SPLINE
SPL {X  -160.133, Y  +702.956, Z    +0.000, E1   -19.806, E3 +400827.881}
SPL {X  -161.979, Y  +690.023, Z    +0.000, E1   -12.991, E3 +400830.798}
SPL {X  -162.641, Y  +681.139, Z    +0.000, E1    -7.893, E3 +400832.889}
SPL {X  -162.815, Y  +674.833, Z    +0.000, E1    -4.093, E3 +400830.505}
SPL {X  -162.820, Y  +669.862, Z    +0.000, E1    -0.751, E3 +400833.723}
SPL {X  -162.820, Y  +665.790, Z    +0.000, E1    +2.338, E3 +400833.096}
SPL {X  -162.820, Y  +660.758, Z    +0.000, E1    +6.523, E3 +400833.197}
SPL {X  -162.820, Y  +655.722, Z    +0.000, E1   +11.608, E3 +400829.570}
SPL {X  -162.820, Y  +648.706, Z    +0.000, E1   +17.761, E3 +400833.112}
SPL {X  -162.820, Y  +635.926, Z    +0.000, E1   +28.192, E3 +400837.939}
SPL {X  -162.820, Y  +621.673, Z    +0.000, E1   +34.265, E3 +400854.297}
SPL {X  -162.820, Y  +609.002, Z    +0.000, E1   +38.458, E3 +400867.518}
SPL {X  -162.820, Y  +596.392, Z    +0.000, E1   +37.895, E3 +400900.987}
ENDSPLINE

SPLINE
SPL {X  -162.820, Y  +601.432, Z    +0.000, E1   +34.026, E3 +400910.285}
ENDSPLINE

SPLINE
SPL {X  -162.820, Y  +597.570, Z    +0.000, E1   +33.919, E3 +400923.183}
SPL {X  -162.820, Y  +592.692, Z    +0.000, E1   +33.779, E3 +400939.074}
SPL {X  -162.820, Y  +588.795, Z    +0.000, E1   +33.876, E3 +400950.511}
SPL {X  -162.820, Y  +585.519, Z    +0.000, E1   +33.888, E3 +400960.596}
SPL {X  -162.820, Y  +582.066, Z    +0.000, E1   +33.857, E3 +400971.530}
SPL {X  -162.820, Y  +577.919, Z    +0.000, E1   +33.841, E3 +400984.583}
SPL {X  -162.820, Y  +573.566, Z    +0.000, E1   +33.899, E3 +400997.658}
SPL {X  -162.820, Y  +569.298, Z    +0.000, E1   +33.851, E3 +401011.300}
SPL {X  -162.820, Y  +565.024, Z    +0.000, E1   +33.872, E3 +401024.355}
SPL {X  -162.820, Y  +560.226, Z    +0.000, E1   +33.868, E3 +401039.449}
SPL {X  -162.820, Y  +556.206, Z    +0.000, E1   +33.843, E3 +401051.849}
SPL {X  -162.820, Y  +553.486, Z    +0.000, E1   +33.777, E3 +401060.795}
SPL {X  -162.820, Y  +549.726, Z    +0.000, E1   +33.905, E3 +401071.650}
SPL {X  -162.820, Y  +545.760, Z    +0.000, E1   +33.901, E3 +401084.046}
SPL {X  -162.820, Y  +541.668, Z    +0.000, E1   +33.787, E3 +401097.446}
SPL {X  -162.820, Y  +537.061, Z    +0.000, E1   +33.897, E3 +401111.104}
SPL {X  -162.820, Y  +532.164, Z    +0.000, E1   +33.861, E3 +401126.578}
SPL {X  -162.820, Y  +528.475, Z    +0.000, E1   +33.876, E3 +401137.746}
SPL {X  -162.820, Y  +524.900, Z    +0.000, E1   +33.820, E3 +401149.405}
SPL {X  -162.820, Y  +520.532, Z    +0.000, E1   +33.805, E3 +401162.973}
SPL {X  -162.820, Y  +515.754, Z    +0.000, E1   +33.911, E3 +401177.309}
SPL {X  -162.820, Y  +510.207, Z    +0.000, E1   +33.879, E3 +401194.689}
SPL {X  -162.820, Y  +504.570, Z    +0.000, E1   +33.876, E3 +401212.269}
SPL {X  -162.820, Y  +498.875, Z    +0.000, E1   +34.747, E3 +401223.970}
SPL {X  -162.820, Y  +481.122, Z    +0.000, E1   +41.279, E3 +401231.121}
SPL {X  -162.820, Y  +477.698, Z    +0.000, E1   +40.353, E3 +401245.177}
SPL {X  -162.820, Y  +473.851, Z    +0.000, E1   +39.059, E3 +401262.569}
SPL {X  -162.820, Y  +470.157, Z    +0.000, E1   +38.016, E3 +401278.506}
SPL {X  -162.820, Y  +467.216, Z    +0.000, E1   +37.215, E3 +401291.267}
SPL {X  -162.820, Y  +462.598, Z    +0.000, E1   +37.325, E3 +401303.221}
SPL {X  -162.820, Y  +459.177, Z    +0.000, E1   +37.207, E3 +401313.249}
SPL {X  -162.820, Y  +453.939, Z    +0.000, E1   +37.397, E3 +401326.601}
SPL {X  -162.820, Y  +448.311, Z    +0.000, E1   +37.333, E3 +401342.262}
SPL {X  -162.820, Y  +443.351, Z    +0.000, E1   +37.335, E3 +401355.792}
SPL {X  -162.820, Y  +438.727, Z    +0.000, E1   +37.289, E3 +401368.664}
SPL {X  -162.820, Y  +434.320, Z    +0.000, E1   +37.343, E3 +401380.374}
SPL {X  -162.820, Y  +430.091, Z    +0.000, E1   +37.424, E3 +401391.374}
SPL {X  -162.820, Y  +426.177, Z    +0.000, E1   +37.250, E3 +401403.197}
SPL {X  -162.820, Y  +420.241, Z    +0.000, E1   +37.355, E3 +401418.903}
SPL {X  -162.820, Y  +415.595, Z    +0.000, E1   +37.375, E3 +401431.243}
SPL {X  -162.820, Y  +411.860, Z    +0.000, E1   +37.402, E3 +401441.346}
SPL {X  -162.820, Y  +407.726, Z    +0.000, E1   +37.291, E3 +401453.294}
SPL {X  -162.820, Y  +403.543, Z    +0.000, E1   +37.305, E3 +401464.639}
SPL {X  -162.820, Y  +399.300, Z    +0.000, E1   +37.355, E3 +401475.924}
SPL {X  -162.820, Y  +395.182, Z    +0.000, E1   +37.347, E3 +401487.213}
SPL {X  -162.820, Y  +390.797, Z    +0.000, E1   +37.358, E3 +401499.125}
SPL {X  -162.820, Y  +386.671, Z    +0.000, E1   +37.363, E3 +401510.306}
SPL {X  -162.820, Y  +382.174, Z    +0.000, E1   +37.329, E3 +401522.883}
SPL {X  -162.785, Y  +377.133, Z    +0.000, E1   +37.299, E3 +401536.813}
SPL {X  -162.576, Y  +371.586, Z    +0.000, E1   +37.322, E3 +401551.925}
SPL {X  -162.256, Y  +366.963, Z    +0.000, E1   +37.251, E3 +401564.814}
SPL {X  -161.920, Y  +363.407, Z    +0.000, E1   +37.164, E3 +401575.099}
SPL {X  -161.341, Y  +358.603, Z    +0.000, E1   +37.117, E3 +401588.579}
SPL {X  -160.616, Y  +353.801, Z    +0.000, E1   +36.942, E3 +401602.744}
SPL {X  -159.837, Y  +349.474, Z    +0.000, E1   +36.824, E3 +401615.188}
SPL {X  -159.171, Y  +346.224, Z    +0.000, E1   +36.747, E3 +401624.464}
SPL {X  -158.248, Y  +342.188, Z    +0.000, E1   +36.583, E3 +401636.627}
SPL {X  -153.520, Y  +326.260, Z    +0.000, E1   +41.363, E3 +401649.279}
SPL {X  -150.942, Y  +319.452, Z    +0.000, E1   +36.529, E3 +401705.636}
ENDSPLINE

SPLINE
SPL {X  -159.264, Y  +346.659, Z    +0.000, E1   +22.083, E3 +401746.211}
SPL {X  -161.245, Y  +357.907, Z    +0.000, E1   +16.095, E3 +401759.643}
SPL {X  -162.697, Y  +374.161, Z    +0.000, E1    +7.119, E3 +401757.633}
SPL {X  -162.820, Y  +380.878, Z    +0.000, E1    +2.854, E3 +401760.464}
SPL {X  -162.820, Y  +385.313, Z    +0.000, E1    -0.228, E3 +401760.244}
SPL {X  -162.820, Y  +389.965, Z    +0.000, E1    -3.918, E3 +401759.613}
SPL {X  -162.820, Y  +394.532, Z    +0.000, E1    -7.849, E3 +401761.161}
SPL {X  -162.820, Y  +400.765, Z    +0.000, E1   -14.108, E3 +401758.628}
SPL {X  -162.820, Y  +411.829, Z    +0.000, E1   -24.195, E3 +401760.705}
SPL {X  -162.820, Y  +434.900, Z    +0.000, E1   -34.666, E3 +401788.070}
SPL {X  -162.820, Y  +465.440, Z    +0.000, E1   -41.264, E3 +401829.377}
ENDSPLINE

SPLINE
SPL {X  -162.820, Y  +460.175, Z    +0.000, E1   -36.098, E3 +401847.177}
ENDSPLINE

SPLINE
SPL {X  -162.820, Y  +465.690, Z    +0.000, E1   -36.140, E3 +401862.491}
SPL {X  -162.820, Y  +470.432, Z    +0.000, E1   -36.100, E3 +401876.374}
SPL {X  -162.820, Y  +475.701, Z    +0.000, E1   -36.157, E3 +401891.001}
SPL {X  -162.820, Y  +479.954, Z    +0.000, E1   -36.086, E3 +401903.542}
SPL {X  -162.820, Y  +485.438, Z    +0.000, E1   -36.112, E3 +401919.260}
SPL {X  -162.820, Y  +490.843, Z    +0.000, E1   -36.087, E3 +401934.673}
SPL {X  -162.820, Y  +494.712, Z    +0.000, E1   -36.164, E3 +401945.185}
SPL {X  -162.820, Y  +497.796, Z    +0.000, E1   -36.022, E3 +401954.891}
SPL {X  -162.820, Y  +502.146, Z    +0.000, E1   -36.123, E3 +401966.760}
SPL {X  -162.820, Y  +505.688, Z    +0.000, E1   -36.050, E3 +401977.242}
SPL {X  -162.820, Y  +509.364, Z    +0.000, E1   -36.084, E3 +401987.613}
SPL {X  -162.820, Y  +513.393, Z    +0.000, E1   -36.179, E3 +401998.469}
SPL {X  -162.820, Y  +516.436, Z    +0.000, E1   -36.094, E3 +402007.665}
SPL {X  -162.820, Y  +520.482, Z    +0.000, E1   -36.096, E3 +402019.296}
SPL {X  -162.820, Y  +524.107, Z    +0.000, E1   -36.045, E3 +402029.880}
SPL {X  -162.820, Y  +527.962, Z    +0.000, E1   -36.074, E3 +402040.813}
SPL {X  -162.820, Y  +532.253, Z    +0.000, E1   -36.170, E3 +402052.402}
SPL {X  -162.820, Y  +536.031, Z    +0.000, E1   -36.058, E3 +402063.940}
SPL {X  -162.820, Y  +541.179, Z    +0.000, E1   -36.085, E3 +402078.581}
SPL {X  -162.820, Y  +546.355, Z    +0.000, E1   -36.114, E3 +402093.125}
SPL {X  -162.820, Y  +551.776, Z    +0.000, E1   -36.108, E3 +402108.759}
SPL {X  -162.820, Y  +558.272, Z    +0.000, E1   -36.170, E3 +402126.967}
SPL {X  -162.820, Y  +562.721, Z    +0.000, E1   -36.046, E3 +402140.192}
SPL {X  -162.820, Y  +566.500, Z    +0.000, E1   -36.073, E3 +402150.924}
SPL {X  -162.820, Y  +570.319, Z    +0.000, E1   -36.045, E3 +402161.953}
SPL {X  -162.820, Y  +573.265, Z    +0.000, E1   -36.071, E3 +402170.189}
SPL {X  -162.820, Y  +576.887, Z    +0.000, E1   -36.084, E3 +402180.547}
SPL {X  -162.820, Y  +581.763, Z    +0.000, E1   -36.093, E3 +402194.484}
SPL {X  -162.820, Y  +586.693, Z    +0.000, E1   -36.086, E3 +402208.589}
SPL {X  -162.820, Y  +591.665, Z    +0.000, E1   -36.045, E3 +402223.117}
SPL {X  -162.820, Y  +597.399, Z    +0.000, E1   -36.147, E3 +402238.880}
SPL {X  -162.820, Y  +602.243, Z    +0.000, E1   -36.085, E3 +402253.026}
SPL {X  -162.820, Y  +605.848, Z    +0.000, E1   -36.070, E3 +402263.348}
SPL {X  -162.820, Y  +609.375, Z    +0.000, E1   -36.084, E3 +402273.398}
SPL {X  -162.820, Y  +612.959, Z    +0.000, E1   -36.034, E3 +402283.918}
SPL {X  -162.820, Y  +616.897, Z    +0.000, E1   -36.061, E3 +402295.066}
SPL {X  -162.820, Y  +621.516, Z    +0.000, E1   -36.072, E3 +402308.265}
SPL {X  -162.820, Y  +626.243, Z    +0.000, E1   -36.105, E3 +402321.508}
SPL {X  -162.820, Y  +630.571, Z    +0.000, E1   -36.057, E3 +402334.210}
SPL {X  -162.820, Y  +634.189, Z    +0.000, E1   -36.065, E3 +402344.403}
SPL {X  -162.820, Y  +638.473, Z    +0.000, E1   -36.098, E3 +402356.640}
SPL {X  -162.820, Y  +642.832, Z    +0.000, E1   -36.091, E3 +402368.966}
SPL {X  -162.820, Y  +646.320, Z    +0.000, E1   -36.078, E3 +402379.073}
SPL {X  -162.820, Y  +649.997, Z    +0.000, E1   -36.000, E3 +402390.044}
SPL {X  -162.820, Y  +655.571, Z    +0.000, E1   -36.141, E3 +402405.378}
SPL {X  -162.820, Y  +661.560, Z    +0.000, E1   -36.068, E3 +402422.806}
SPL {X  -162.820, Y  +667.641, Z    +0.000, E1   -36.092, E3 +402440.187}
SPL {X  -162.820, Y  +673.415, Z    +0.000, E1   -36.053, E3 +402456.777}
SPL {X  -162.761, Y  +677.889, Z    +0.000, E1   -36.122, E3 +402469.095}
SPL {X  -162.577, Y  +682.401, Z    +0.000, E1   -36.021, E3 +402482.712}
SPL {X  -162.187, Y  +687.846, Z    +0.000, E1   -36.007, E3 +402498.381}
SPL {X  -161.667, Y  +692.839, Z    +0.000, E1   -35.918, E3 +402513.146}
SPL {X  -161.078, Y  +697.256, Z    +0.000, E1   -35.797, E3 +402526.482}
SPL {X  -160.313, Y  +701.964, Z    +0.000, E1   -35.709, E3 +402540.558}
SPL {X  -159.317, Y  +707.091, Z    +0.000, E1   -35.482, E3 +402556.582}
SPL {X  -158.510, Y  +710.714, Z    +0.000, E1   -35.230, E3 +402568.293}
SPL {X  -155.037, Y  +723.239, Z    +0.000, E1   -39.382, E3 +402577.389}
SPL {X  -152.141, Y  +731.494, Z    +0.000, E1   -35.181, E3 +402636.195}
ENDSPLINE

SPLINE
SPL {X  -160.133, Y  +702.956, Z    +0.000, E1   -19.806, E3 +402679.733}
SPL {X  -161.979, Y  +690.023, Z    +0.000, E1   -12.991, E3 +402682.649}
SPL {X  -162.641, Y  +681.139, Z    +0.000, E1    -7.893, E3 +402684.741}
SPL {X  -162.815, Y  +674.833, Z    +0.000, E1    -4.093, E3 +402682.357}
SPL {X  -162.820, Y  +669.862, Z    +0.000, E1    -0.751, E3 +402685.575}
SPL {X  -162.820, Y  +664.572, Z    +0.000, E1    +3.252, E3 +402685.389}
SPL {X  -162.820, Y  +657.781, Z    +0.000, E1    +9.391, E3 +402683.212}
SPL {X  -162.820, Y  +648.706, Z    +0.000, E1   +17.761, E3 +402684.964}
SPL {X  -162.820, Y  +635.926, Z    +0.000, E1   +28.192, E3 +402689.791}
SPL {X  -162.820, Y  +621.673, Z    +0.000, E1   +34.265, E3 +402706.149}
SPL {X  -162.820, Y  +601.185, Z    +0.000, E1   +39.430, E3 +402732.727}
SPL {X  -162.820, Y  +599.927, Z    +0.000, E1   +35.241, E3 +402759.305}
SPL {X  -162.820, Y  +597.570, Z    +0.000, E1   +33.919, E3 +402775.034}
SPL {X  -162.820, Y  +592.692, Z    +0.000, E1   +33.779, E3 +402790.926}
SPL {X  -162.820, Y  +588.795, Z    +0.000, E1   +33.876, E3 +402802.363}
SPL {X  -162.820, Y  +584.646, Z    +0.000, E1   +33.882, E3 +402815.327}
SPL {X  -162.820, Y  +579.919, Z    +0.000, E1   +33.857, E3 +402830.115}
SPL {X  -162.820, Y  +574.615, Z    +0.000, E1   +33.920, E3 +402846.289}
SPL {X  -162.820, Y  +570.335, Z    +0.000, E1   +33.821, E3 +402859.995}
SPL {X  -162.820, Y  +565.901, Z    +0.000, E1   +33.889, E3 +402873.515}
SPL {X  -162.820, Y  +562.173, Z    +0.000, E1   +33.897, E3 +402884.806}
SPL {X  -162.820, Y  +558.179, Z    +0.000, E1   +33.857, E3 +402897.742}
SPL {X  -162.820, Y  +553.486, Z    +0.000, E1   +33.777, E3 +402912.647}
SPL {X  -162.820, Y  +548.576, Z    +0.000, E1   +33.950, E3 +402926.929}
SPL {X  -162.820, Y  +544.808, Z    +0.000, E1   +33.827, E3 +402939.191}
SPL {X  -162.820, Y  +541.668, Z    +0.000, E1   +33.787, E3 +402949.297}
SPL {X  -162.820, Y  +538.174, Z    +0.000, E1   +33.865, E3 +402959.587}
SPL {X  -162.820, Y  +534.943, Z    +0.000, E1   +33.919, E3 +402969.327}
SPL {X  -162.820, Y  +531.459, Z    +0.000, E1   +33.783, E3 +402980.984}
SPL {X  -162.820, Y  +528.475, Z    +0.000, E1   +33.876, E3 +402989.598}
SPL {X  -162.820, Y  +524.900, Z    +0.000, E1   +33.820, E3 +403001.257}
SPL {X  -162.820, Y  +520.532, Z    +0.000, E1   +33.805, E3 +403014.825}
SPL {X  -162.820, Y  +516.814, Z    +0.000, E1   +33.917, E3 +403025.661}
SPL {X  -162.820, Y  +512.685, Z    +0.000, E1   +33.830, E3 +403039.103}
SPL {X  -162.820, Y  +508.888, Z    +0.000, E1   +33.871, E3 +403050.518}
SPL {X  -162.820, Y  +505.651, Z    +0.000, E1   +33.839, E3 +403060.835}
SPL {X  -162.820, Y  +500.931, Z    +0.000, E1   +34.256, E3 +403072.709}
SPL {X  -162.820, Y  +481.122, Z    +0.000, E1   +41.279, E3 +403082.973}
SPL {X  -162.820, Y  +477.698, Z    +0.000, E1   +40.353, E3 +403097.029}
SPL {X  -162.820, Y  +474.538, Z    +0.000, E1   +39.267, E3 +403111.205}
SPL {X  -162.820, Y  +472.097, Z    +0.000, E1   +38.411, E3 +403122.748}
SPL {X  -162.820, Y  +469.308, Z    +0.000, E1   +37.839, E3 +403133.553}
SPL {X  -162.820, Y  +467.216, Z    +0.000, E1   +37.215, E3 +403143.119}
SPL {X  -162.820, Y  +462.598, Z    +0.000, E1   +37.325, E3 +403155.073}
SPL {X  -162.820, Y  +457.832, Z    +0.000, E1   +37.294, E3 +403168.360}
SPL {X  -162.820, Y  +452.986, Z    +0.000, E1   +37.368, E3 +403181.094}
SPL {X  -162.820, Y  +448.311, Z    +0.000, E1   +37.333, E3 +403194.114}
SPL {X  -162.820, Y  +443.351, Z    +0.000, E1   +37.335, E3 +403207.643}
SPL {X  -162.820, Y  +438.727, Z    +0.000, E1   +37.289, E3 +403220.516}
SPL {X  -162.820, Y  +434.320, Z    +0.000, E1   +37.343, E3 +403232.226}
SPL {X  -162.820, Y  +430.091, Z    +0.000, E1   +37.424, E3 +403243.226}
SPL {X  -162.820, Y  +426.177, Z    +0.000, E1   +37.250, E3 +403255.048}
SPL {X  -162.820, Y  +421.391, Z    +0.000, E1   +37.346, E3 +403267.512}
SPL {X  -162.820, Y  +416.811, Z    +0.000, E1   +37.348, E3 +403280.046}
SPL {X  -162.820, Y  +411.860, Z    +0.000, E1   +37.402, E3 +403293.198}
SPL {X  -162.820, Y  +407.726, Z    +0.000, E1   +37.291, E3 +403305.146}
SPL {X  -162.820, Y  +403.543, Z    +0.000, E1   +37.305, E3 +403316.491}
SPL {X  -162.820, Y  +399.300, Z    +0.000, E1   +37.355, E3 +403327.776}
SPL {X  -162.820, Y  +395.182, Z    +0.000, E1   +37.347, E3 +403339.065}
SPL {X  -162.820, Y  +390.797, Z    +0.000, E1   +37.358, E3 +403350.977}
SPL {X  -162.820, Y  +385.307, Z    +0.000, E1   +37.364, E3 +403366.057}
SPL {X  -162.820, Y  +380.796, Z    +0.000, E1   +37.334, E3 +403378.343}
SPL {X  -162.785, Y  +377.133, Z    +0.000, E1   +37.299, E3 +403388.664}
SPL {X  -162.623, Y  +372.484, Z    +0.000, E1   +37.337, E3 +403401.104}
SPL {X  -162.331, Y  +367.894, Z    +0.000, E1   +37.251, E3 +403414.217}
SPL {X  -161.920, Y  +363.407, Z    +0.000, E1   +37.164, E3 +403426.951}
SPL {X  -161.341, Y  +358.603, Z    +0.000, E1   +37.117, E3 +403440.431}
SPL {X  -160.616, Y  +353.801, Z    +0.000, E1   +36.942, E3 +403454.595}
SPL {X  -159.837, Y  +349.474, Z    +0.000, E1   +36.824, E3 +403467.040}
SPL {X  -158.862, Y  +344.820, Z    +0.000, E1   +36.732, E3 +403480.402}
SPL {X  -157.959, Y  +341.011, Z    +0.000, E1   +36.448, E3 +403492.299}
SPL {X  -154.495, Y  +329.104, Z    +0.000, E1   +40.891, E3 +403497.182}
SPL {X  -152.543, Y  +323.569, Z    +0.000, E1   +41.772, E3 +403504.938}
SPL {X  -150.942, Y  +319.452, Z    +0.000, E1   +36.529, E3 +403557.488}
ENDSPLINE

SPLINE
SPL {X  -159.264, Y  +346.659, Z    +0.000, E1   +22.083, E3 +403598.062}
SPL {X  -161.245, Y  +357.907, Z    +0.000, E1   +16.095, E3 +403611.495}
SPL {X  -162.697, Y  +374.161, Z    +0.000, E1    +7.119, E3 +403609.485}
SPL {X  -162.820, Y  +380.878, Z    +0.000, E1    +2.854, E3 +403612.316}
SPL {X  -162.820, Y  +385.313, Z    +0.000, E1    -0.228, E3 +403612.096}
SPL {X  -162.820, Y  +389.965, Z    +0.000, E1    -3.918, E3 +403611.465}
SPL {X  -162.820, Y  +394.532, Z    +0.000, E1    -7.849, E3 +403613.013}
SPL {X  -162.820, Y  +400.765, Z    +0.000, E1   -14.108, E3 +403610.480}
SPL {X  -162.820, Y  +411.829, Z    +0.000, E1   -24.195, E3 +403612.557}
SPL {X  -162.820, Y  +434.900, Z    +0.000, E1   -34.666, E3 +403639.922}
SPL {X  -162.820, Y  +465.440, Z    +0.000, E1   -41.264, E3 +403681.229}
ENDSPLINE

SPLINE
SPL {X  -162.820, Y  +460.175, Z    +0.000, E1   -36.098, E3 +403699.029}
ENDSPLINE

SPLINE
SPL {X  -162.820, Y  +465.690, Z    +0.000, E1   -36.140, E3 +403714.343}
SPL {X  -162.820, Y  +470.432, Z    +0.000, E1   -36.100, E3 +403728.226}
SPL {X  -162.820, Y  +475.701, Z    +0.000, E1   -36.157, E3 +403742.853}
SPL {X  -162.820, Y  +479.954, Z    +0.000, E1   -36.086, E3 +403755.393}
SPL {X  -162.820, Y  +485.438, Z    +0.000, E1   -36.112, E3 +403771.112}
SPL {X  -162.820, Y  +490.843, Z    +0.000, E1   -36.087, E3 +403786.525}
SPL {X  -162.820, Y  +494.712, Z    +0.000, E1   -36.164, E3 +403797.037}
SPL {X  -162.820, Y  +497.796, Z    +0.000, E1   -36.022, E3 +403806.743}
SPL {X  -162.820, Y  +502.146, Z    +0.000, E1   -36.123, E3 +403818.612}
SPL {X  -162.820, Y  +505.688, Z    +0.000, E1   -36.050, E3 +403829.094}
SPL {X  -162.820, Y  +509.364, Z    +0.000, E1   -36.084, E3 +403839.465}
SPL {X  -162.820, Y  +513.393, Z    +0.000, E1   -36.179, E3 +403850.321}
SPL {X  -162.820, Y  +516.436, Z    +0.000, E1   -36.094, E3 +403859.517}
SPL {X  -162.820, Y  +520.482, Z    +0.000, E1   -36.096, E3 +403871.148}
SPL {X  -162.820, Y  +524.107, Z    +0.000, E1   -36.045, E3 +403881.732}
SPL {X  -162.820, Y  +527.962, Z    +0.000, E1   -36.074, E3 +403892.665}
SPL {X  -162.820, Y  +532.253, Z    +0.000, E1   -36.170, E3 +403904.254}
SPL {X  -162.820, Y  +536.031, Z    +0.000, E1   -36.058, E3 +403915.792}
SPL {X  -162.820, Y  +541.179, Z    +0.000, E1   -36.085, E3 +403930.433}
SPL {X  -162.820, Y  +546.355, Z    +0.000, E1   -36.114, E3 +403944.977}
SPL {X  -162.820, Y  +551.776, Z    +0.000, E1   -36.108, E3 +403960.611}
SPL {X  -162.820, Y  +558.272, Z    +0.000, E1   -36.170, E3 +403978.819}
SPL {X  -162.820, Y  +562.721, Z    +0.000, E1   -36.046, E3 +403992.044}
SPL {X  -162.820, Y  +566.500, Z    +0.000, E1   -36.073, E3 +404002.776}
SPL {X  -162.820, Y  +570.319, Z    +0.000, E1   -36.045, E3 +404013.804}
SPL {X  -162.820, Y  +573.265, Z    +0.000, E1   -36.071, E3 +404022.041}
SPL {X  -162.820, Y  +576.887, Z    +0.000, E1   -36.084, E3 +404032.399}
SPL {X  -162.820, Y  +581.763, Z    +0.000, E1   -36.093, E3 +404046.336}
SPL {X  -162.820, Y  +586.693, Z    +0.000, E1   -36.086, E3 +404060.441}
SPL {X  -162.820, Y  +591.665, Z    +0.000, E1   -36.045, E3 +404074.969}
SPL {X  -162.820, Y  +597.399, Z    +0.000, E1   -36.147, E3 +404090.732}
SPL {X  -162.820, Y  +602.243, Z    +0.000, E1   -36.085, E3 +404104.878}
SPL {X  -162.820, Y  +605.848, Z    +0.000, E1   -36.070, E3 +404115.199}
SPL {X  -162.820, Y  +609.375, Z    +0.000, E1   -36.084, E3 +404125.250}
SPL {X  -162.820, Y  +612.959, Z    +0.000, E1   -36.034, E3 +404135.770}
SPL {X  -162.820, Y  +616.897, Z    +0.000, E1   -36.061, E3 +404146.918}
SPL {X  -162.820, Y  +621.516, Z    +0.000, E1   -36.072, E3 +404160.117}
SPL {X  -162.820, Y  +626.243, Z    +0.000, E1   -36.105, E3 +404173.360}
SPL {X  -162.820, Y  +630.571, Z    +0.000, E1   -36.057, E3 +404186.062}
SPL {X  -162.820, Y  +634.189, Z    +0.000, E1   -36.065, E3 +404196.255}
SPL {X  -162.820, Y  +638.473, Z    +0.000, E1   -36.098, E3 +404208.492}
SPL {X  -162.820, Y  +642.832, Z    +0.000, E1   -36.091, E3 +404220.818}
SPL {X  -162.820, Y  +646.320, Z    +0.000, E1   -36.078, E3 +404230.925}
SPL {X  -162.820, Y  +649.997, Z    +0.000, E1   -36.000, E3 +404241.896}
SPL {X  -162.820, Y  +655.571, Z    +0.000, E1   -36.141, E3 +404257.230}
SPL {X  -162.820, Y  +661.560, Z    +0.000, E1   -36.068, E3 +404274.658}
SPL {X  -162.820, Y  +667.641, Z    +0.000, E1   -36.092, E3 +404292.039}
SPL {X  -162.820, Y  +673.415, Z    +0.000, E1   -36.053, E3 +404308.629}
SPL {X  -162.761, Y  +677.889, Z    +0.000, E1   -36.122, E3 +404320.947}
SPL {X  -162.577, Y  +682.401, Z    +0.000, E1   -36.021, E3 +404334.564}
SPL {X  -162.187, Y  +687.846, Z    +0.000, E1   -36.007, E3 +404350.233}
SPL {X  -161.667, Y  +692.839, Z    +0.000, E1   -35.918, E3 +404364.998}
SPL {X  -161.078, Y  +697.256, Z    +0.000, E1   -35.797, E3 +404378.334}
SPL {X  -160.313, Y  +701.964, Z    +0.000, E1   -35.709, E3 +404392.410}
SPL {X  -159.317, Y  +707.091, Z    +0.000, E1   -35.482, E3 +404408.433}
SPL {X  -158.510, Y  +710.714, Z    +0.000, E1   -35.230, E3 +404420.144}
SPL {X  -155.037, Y  +723.239, Z    +0.000, E1   -39.382, E3 +404429.241}
SPL {X  -152.141, Y  +731.494, Z    +0.000, E1   -35.181, E3 +404488.047}
ENDSPLINE

SPLINE
SPL {X  -152.670, Y  +730.088, Z    +0.000, E1   -30.916, E3 +404561.409}
SPL {X  -160.727, Y  +699.521, Z    +0.000, E1   -18.202, E3 +404527.692}
SPL {X  -161.979, Y  +690.023, Z    +0.000, E1   -12.991, E3 +404534.501}
SPL {X  -162.641, Y  +681.139, Z    +0.000, E1    -7.893, E3 +404536.593}
SPL {X  -162.820, Y  +673.062, Z    +0.000, E1    -2.992, E3 +404535.560}
SPL {X  -162.820, Y  +666.731, Z    +0.000, E1    +1.545, E3 +404537.190}
SPL {X  -162.820, Y  +660.758, Z    +0.000, E1    +6.523, E3 +404536.901}
SPL {X  -162.820, Y  +650.583, Z    +0.000, E1   +16.035, E3 +404535.873}
SPL {X  -162.820, Y  +629.267, Z    +0.000, E1   +31.872, E3 +404547.022}
SPL {X  -162.820, Y  +617.390, Z    +0.000, E1   +35.413, E3 +404563.951}
SPL {X  -162.820, Y  +596.392, Z    +0.000, E1   +37.895, E3 +404604.691}
ENDSPLINE

SPLINE
SPL {X  -162.820, Y  +601.432, Z    +0.000, E1   +34.026, E3 +404613.989}
ENDSPLINE

SPLINE
SPL {X  -162.820, Y  +597.570, Z    +0.000, E1   +33.919, E3 +404626.886}
SPL {X  -162.820, Y  +592.692, Z    +0.000, E1   +33.779, E3 +404642.778}
SPL {X  -162.820, Y  +588.795, Z    +0.000, E1   +33.876, E3 +404654.215}
SPL {X  -162.820, Y  +585.519, Z    +0.000, E1   +33.888, E3 +404664.300}
SPL {X  -162.820, Y  +582.066, Z    +0.000, E1   +33.857, E3 +404675.234}
SPL {X  -162.820, Y  +577.919, Z    +0.000, E1   +33.841, E3 +404688.287}
SPL {X  -162.820, Y  +573.566, Z    +0.000, E1   +33.899, E3 +404701.362}
SPL {X  -162.820, Y  +569.298, Z    +0.000, E1   +33.851, E3 +404715.003}
SPL {X  -162.820, Y  +563.983, Z    +0.000, E1   +33.916, E3 +404731.144}
SPL {X  -162.820, Y  +559.395, Z    +0.000, E1   +33.796, E3 +404746.025}
SPL {X  -162.820, Y  +554.453, Z    +0.000, E1   +33.841, E3 +404761.250}
SPL {X  -162.820, Y  +549.726, Z    +0.000, E1   +33.905, E3 +404775.353}
SPL {X  -162.820, Y  +545.760, Z    +0.000, E1   +33.901, E3 +404787.749}
SPL {X  -162.820, Y  +541.668, Z    +0.000, E1   +33.787, E3 +404801.149}
SPL {X  -162.820, Y  +538.174, Z    +0.000, E1   +33.865, E3 +404811.439}
SPL {X  -162.820, Y  +534.943, Z    +0.000, E1   +33.919, E3 +404821.179}
SPL {X  -162.820, Y  +530.273, Z    +0.000, E1   +33.855, E3 +404836.208}
SPL {X  -162.820, Y  +524.900, Z    +0.000, E1   +33.820, E3 +404853.109}
SPL {X  -162.820, Y  +520.532, Z    +0.000, E1   +33.805, E3 +404866.677}
SPL {X  -162.820, Y  +516.814, Z    +0.000, E1   +33.917, E3 +404877.513}
SPL {X  -162.820, Y  +512.685, Z    +0.000, E1   +33.830, E3 +404890.955}
SPL {X  -162.820, Y  +508.888, Z    +0.000, E1   +33.871, E3 +404902.370}
SPL {X  -162.820, Y  +505.651, Z    +0.000, E1   +33.839, E3 +404912.687}
SPL {X  -162.820, Y  +500.931, Z    +0.000, E1   +34.256, E3 +404924.561}
SPL {X  -162.820, Y  +481.122, Z    +0.000, E1   +41.279, E3 +404934.825}
SPL {X  -162.820, Y  +477.698, Z    +0.000, E1   +40.353, E3 +404948.881}
SPL {X  -162.820, Y  +474.538, Z    +0.000, E1   +39.267, E3 +404963.056}
SPL {X  -162.820, Y  +472.097, Z    +0.000, E1   +38.411, E3 +404974.600}
SPL {X  -162.820, Y  +469.308, Z    +0.000, E1   +37.839, E3 +404985.404}
SPL {X  -162.820, Y  +467.216, Z    +0.000, E1   +37.215, E3 +404994.971}
SPL {X  -162.820, Y  +462.598, Z    +0.000, E1   +37.325, E3 +405006.925}
SPL {X  -162.820, Y  +457.832, Z    +0.000, E1   +37.294, E3 +405020.212}
SPL {X  -162.820, Y  +452.986, Z    +0.000, E1   +37.368, E3 +405032.946}
SPL {X  -162.820, Y  +448.311, Z    +0.000, E1   +37.333, E3 +405045.966}
SPL {X  -162.820, Y  +443.351, Z    +0.000, E1   +37.335, E3 +405059.495}
SPL {X  -162.820, Y  +438.727, Z    +0.000, E1   +37.289, E3 +405072.368}
SPL {X  -162.820, Y  +434.320, Z    +0.000, E1   +37.343, E3 +405084.078}
SPL {X  -162.820, Y  +430.091, Z    +0.000, E1   +37.424, E3 +405095.078}
SPL {X  -162.820, Y  +426.177, Z    +0.000, E1   +37.250, E3 +405106.900}
SPL {X  -162.820, Y  +421.391, Z    +0.000, E1   +37.346, E3 +405119.364}
SPL {X  -162.820, Y  +416.811, Z    +0.000, E1   +37.348, E3 +405131.898}
SPL {X  -162.820, Y  +411.860, Z    +0.000, E1   +37.402, E3 +405145.050}
SPL {X  -162.820, Y  +407.726, Z    +0.000, E1   +37.291, E3 +405156.998}
SPL {X  -162.820, Y  +403.543, Z    +0.000, E1   +37.305, E3 +405168.343}
SPL {X  -162.820, Y  +399.300, Z    +0.000, E1   +37.355, E3 +405179.627}
SPL {X  -162.820, Y  +395.182, Z    +0.000, E1   +37.347, E3 +405190.917}
SPL {X  -162.820, Y  +390.797, Z    +0.000, E1   +37.358, E3 +405202.829}
SPL {X  -162.820, Y  +385.307, Z    +0.000, E1   +37.364, E3 +405217.908}
SPL {X  -162.820, Y  +380.796, Z    +0.000, E1   +37.334, E3 +405230.195}
SPL {X  -162.785, Y  +377.133, Z    +0.000, E1   +37.299, E3 +405240.516}
SPL {X  -162.623, Y  +372.484, Z    +0.000, E1   +37.337, E3 +405252.956}
SPL {X  -162.331, Y  +367.894, Z    +0.000, E1   +37.251, E3 +405266.069}
SPL {X  -161.920, Y  +363.407, Z    +0.000, E1   +37.164, E3 +405278.803}
SPL {X  -161.341, Y  +358.603, Z    +0.000, E1   +37.117, E3 +405292.283}
SPL {X  -160.616, Y  +353.801, Z    +0.000, E1   +36.942, E3 +405306.447}
SPL {X  -159.837, Y  +349.474, Z    +0.000, E1   +36.824, E3 +405318.891}
SPL {X  -158.862, Y  +344.820, Z    +0.000, E1   +36.732, E3 +405332.254}
SPL {X  -157.959, Y  +341.011, Z    +0.000, E1   +36.448, E3 +405344.151}
SPL {X  -154.495, Y  +329.104, Z    +0.000, E1   +40.891, E3 +405349.033}
SPL {X  -152.543, Y  +323.569, Z    +0.000, E1   +41.772, E3 +405356.790}
SPL {X  -150.942, Y  +319.452, Z    +0.000, E1   +36.529, E3 +405409.340}
ENDSPLINE

SPLINE
SPL {X  -159.264, Y  +346.659, Z    +0.000, E1   +22.083, E3 +405449.914}
SPL {X  -161.245, Y  +357.907, Z    +0.000, E1   +16.095, E3 +405463.347}
SPL {X  -162.746, Y  +375.590, Z    +0.000, E1    +6.280, E3 +405462.935}
SPL {X  -162.820, Y  +384.478, Z    +0.000, E1    +0.434, E3 +405463.605}
SPL {X  -162.820, Y  +389.965, Z    +0.000, E1    -3.918, E3 +405463.316}
SPL {X  -162.820, Y  +394.532, Z    +0.000, E1    -7.849, E3 +405464.865}
SPL {X  -162.820, Y  +400.765, Z    +0.000, E1   -14.108, E3 +405462.331}
SPL {X  -162.820, Y  +411.829, Z    +0.000, E1   -24.195, E3 +405464.409}
SPL {X  -162.820, Y  +434.900, Z    +0.000, E1   -34.666, E3 +405491.774}
SPL {X  -162.820, Y  +465.440, Z    +0.000, E1   -41.264, E3 +405533.081}
ENDSPLINE

SPLINE
SPL {X  -162.820, Y  +460.175, Z    +0.000, E1   -36.098, E3 +405550.881}
ENDSPLINE

SPLINE
SPL {X  -162.820, Y  +465.690, Z    +0.000, E1   -36.140, E3 +405566.195}
SPL {X  -162.820, Y  +470.432, Z    +0.000, E1   -36.100, E3 +405580.077}
SPL {X  -162.820, Y  +475.701, Z    +0.000, E1   -36.157, E3 +405594.705}
SPL {X  -162.820, Y  +479.954, Z    +0.000, E1   -36.086, E3 +405607.245}
SPL {X  -162.820, Y  +483.976, Z    +0.000, E1   -36.049, E3 +405618.977}
SPL {X  -162.820, Y  +488.601, Z    +0.000, E1   -36.081, E3 +405632.067}
SPL {X  -162.820, Y  +493.837, Z    +0.000, E1   -36.178, E3 +405646.411}
SPL {X  -162.820, Y  +497.796, Z    +0.000, E1   -36.022, E3 +405658.595}
SPL {X  -162.820, Y  +502.146, Z    +0.000, E1   -36.123, E3 +405670.464}
SPL {X  -162.820, Y  +505.688, Z    +0.000, E1   -36.050, E3 +405680.946}
SPL {X  -162.820, Y  +509.364, Z    +0.000, E1   -36.084, E3 +405691.317}
SPL {X  -162.820, Y  +513.393, Z    +0.000, E1   -36.179, E3 +405702.173}
SPL {X  -162.820, Y  +516.436, Z    +0.000, E1   -36.094, E3 +405711.368}
SPL {X  -162.820, Y  +520.482, Z    +0.000, E1   -36.096, E3 +405723.000}
SPL {X  -162.820, Y  +524.107, Z    +0.000, E1   -36.045, E3 +405733.584}
SPL {X  -162.820, Y  +527.962, Z    +0.000, E1   -36.074, E3 +405744.517}
SPL {X  -162.820, Y  +532.253, Z    +0.000, E1   -36.170, E3 +405756.106}
SPL {X  -162.820, Y  +536.031, Z    +0.000, E1   -36.058, E3 +405767.644}
SPL {X  -162.820, Y  +541.179, Z    +0.000, E1   -36.085, E3 +405782.285}
SPL {X  -162.820, Y  +546.355, Z    +0.000, E1   -36.114, E3 +405796.829}
SPL {X  -162.820, Y  +551.776, Z    +0.000, E1   -36.108, E3 +405812.463}
SPL {X  -162.820, Y  +556.944, Z    +0.000, E1   -36.118, E3 +405827.033}
SPL {X  -162.820, Y  +561.684, Z    +0.000, E1   -36.118, E3 +405840.625}
SPL {X  -162.820, Y  +566.500, Z    +0.000, E1   -36.073, E3 +405854.628}
SPL {X  -162.820, Y  +571.734, Z    +0.000, E1   -36.094, E3 +405869.558}
SPL {X  -162.820, Y  +576.887, Z    +0.000, E1   -36.084, E3 +405884.251}
SPL {X  -162.820, Y  +581.763, Z    +0.000, E1   -36.093, E3 +405898.188}
SPL {X  -162.820, Y  +586.693, Z    +0.000, E1   -36.086, E3 +405912.293}
SPL {X  -162.820, Y  +590.250, Z    +0.000, E1   -36.075, E3 +405922.412}
SPL {X  -162.820, Y  +592.727, Z    +0.000, E1   -35.960, E3 +405930.236}
SPL {X  -162.820, Y  +597.399, Z    +0.000, E1   -36.147, E3 +405942.584}
SPL {X  -162.820, Y  +602.243, Z    +0.000, E1   -36.085, E3 +405956.730}
SPL {X  -162.820, Y  +606.975, Z    +0.000, E1   -36.102, E3 +405970.175}
SPL {X  -162.820, Y  +611.980, Z    +0.000, E1   -36.072, E3 +405984.721}
SPL {X  -162.820, Y  +616.897, Z    +0.000, E1   -36.061, E3 +405998.770}
SPL {X  -162.820, Y  +621.516, Z    +0.000, E1   -36.072, E3 +406011.969}
SPL {X  -162.820, Y  +626.243, Z    +0.000, E1   -36.105, E3 +406025.211}
SPL {X  -162.820, Y  +630.571, Z    +0.000, E1   -36.057, E3 +406037.913}
SPL {X  -162.820, Y  +634.189, Z    +0.000, E1   -36.065, E3 +406048.107}
SPL {X  -162.820, Y  +638.473, Z    +0.000, E1   -36.098, E3 +406060.344}
SPL {X  -162.820, Y  +642.832, Z    +0.000, E1   -36.091, E3 +406072.670}
SPL {X  -162.820, Y  +646.320, Z    +0.000, E1   -36.078, E3 +406082.777}
SPL {X  -162.820, Y  +649.997, Z    +0.000, E1   -36.000, E3 +406093.748}
SPL {X  -162.820, Y  +655.571, Z    +0.000, E1   -36.141, E3 +406109.082}
SPL {X  -162.820, Y  +661.560, Z    +0.000, E1   -36.068, E3 +406126.509}
SPL {X  -162.820, Y  +666.386, Z    +0.000, E1   -36.048, E3 +406140.394}
SPL {X  -162.820, Y  +672.345, Z    +0.000, E1   -36.097, E3 +406157.334}
SPL {X  -162.761, Y  +677.889, Z    +0.000, E1   -36.122, E3 +406172.799}
SPL {X  -162.577, Y  +682.401, Z    +0.000, E1   -36.021, E3 +406186.416}
SPL {X  -162.296, Y  +686.558, Z    +0.000, E1   -35.952, E3 +406198.606}
SPL {X  -161.948, Y  +690.331, Z    +0.000, E1   -35.960, E3 +406209.404}
SPL {X  -161.544, Y  +693.846, Z    +0.000, E1   -35.908, E3 +406219.680}
SPL {X  -160.925, Y  +698.267, Z    +0.000, E1   -35.816, E3 +406233.112}
SPL {X  -160.151, Y  +702.861, Z    +0.000, E1   -35.643, E3 +406247.082}
SPL {X  -159.317, Y  +707.091, Z    +0.000, E1   -35.482, E3 +406260.285}
SPL {X  -158.510, Y  +710.714, Z    +0.000, E1   -35.230, E3 +406271.996}
SPL {X  -155.037, Y  +723.239, Z    +0.000, E1   -39.382, E3 +406281.093}
SPL {X  -152.141, Y  +731.494, Z    +0.000, E1   -35.181, E3 +406339.898}
ENDSPLINE

SPLINE
SPL {X  -160.133, Y  +702.956, Z    +0.000, E1   -19.806, E3 +406383.436}
SPL {X  -161.979, Y  +690.023, Z    +0.000, E1   -12.991, E3 +406386.353}
SPL {X  -162.641, Y  +681.139, Z    +0.000, E1    -7.893, E3 +406388.445}
SPL {X  -162.815, Y  +674.833, Z    +0.000, E1    -4.093, E3 +406386.061}
SPL {X  -162.820, Y  +669.862, Z    +0.000, E1    -0.751, E3 +406389.279}
SPL {X  -162.820, Y  +664.572, Z    +0.000, E1    +3.252, E3 +406389.093}
SPL {X  -162.820, Y  +657.781, Z    +0.000, E1    +9.391, E3 +406386.916}
SPL {X  -162.820, Y  +648.706, Z    +0.000, E1   +17.761, E3 +406388.667}
SPL {X  -162.820, Y  +635.926, Z    +0.000, E1   +28.192, E3 +406393.495}
SPL {X  -162.820, Y  +621.673, Z    +0.000, E1   +34.265, E3 +406409.852}
SPL {X  -162.820, Y  +609.002, Z    +0.000, E1   +38.458, E3 +406423.074}
SPL {X  -162.820, Y  +596.392, Z    +0.000, E1   +37.895, E3 +406456.543}
ENDSPLINE

SPLINE
SPL {X  -162.820, Y  +601.432, Z    +0.000, E1   +34.026, E3 +406465.841}
ENDSPLINE

SPLINE
SPL {X  -162.820, Y  +599.021, Z    +0.000, E1   +33.912, E3 +406474.059}
SPL {X  -162.820, Y  +595.170, Z    +0.000, E1   +33.784, E3 +406486.965}
SPL {X  -162.820, Y  +589.785, Z    +0.000, E1   +33.904, E3 +406502.962}
SPL {X  -162.820, Y  +585.519, Z    +0.000, E1   +33.888, E3 +406516.152}
SPL {X  -162.820, Y  +580.762, Z    +0.000, E1   +33.875, E3 +406531.229}
SPL {X  -162.820, Y  +574.615, Z    +0.000, E1   +33.920, E3 +406549.993}
SPL {X  -162.820, Y  +569.298, Z    +0.000, E1   +33.851, E3 +406566.855}
SPL {X  -162.820, Y  +565.024, Z    +0.000, E1   +33.872, E3 +406579.911}
SPL {X  -162.820, Y  +560.226, Z    +0.000, E1   +33.868, E3 +406595.004}
SPL {X  -162.820, Y  +556.206, Z    +0.000, E1   +33.843, E3 +406607.404}
SPL {X  -162.820, Y  +553.486, Z    +0.000, E1   +33.777, E3 +406616.351}
SPL {X  -162.820, Y  +548.576, Z    +0.000, E1   +33.950, E3 +406630.632}
SPL {X  -162.820, Y  +544.808, Z    +0.000, E1   +33.827, E3 +406642.895}
SPL {X  -162.820, Y  +541.668, Z    +0.000, E1   +33.787, E3 +406653.001}
SPL {X  -162.820, Y  +538.174, Z    +0.000, E1   +33.865, E3 +406663.291}
SPL {X  -162.820, Y  +534.943, Z    +0.000, E1   +33.919, E3 +406673.031}
SPL {X  -162.820, Y  +530.273, Z    +0.000, E1   +33.855, E3 +406688.060}
SPL {X  -162.820, Y  +524.900, Z    +0.000, E1   +33.820, E3 +406704.961}
SPL {X  -162.820, Y  +520.532, Z    +0.000, E1   +33.805, E3 +406718.528}
SPL {X  -162.820, Y  +516.814, Z    +0.000, E1   +33.917, E3 +406729.364}
SPL {X  -162.820, Y  +512.685, Z    +0.000, E1   +33.830, E3 +406742.807}
SPL {X  -162.820, Y  +508.888, Z    +0.000, E1   +33.871, E3 +406754.222}
SPL {X  -162.820, Y  +505.651, Z    +0.000, E1   +33.839, E3 +406764.539}
SPL {X  -162.820, Y  +500.931, Z    +0.000, E1   +34.256, E3 +406776.412}
SPL {X  -162.820, Y  +481.122, Z    +0.000, E1   +41.279, E3 +406786.677}
SPL {X  -162.820, Y  +478.698, Z    +0.000, E1   +40.526, E3 +406797.026}
SPL {X  -162.820, Y  +476.364, Z    +0.000, E1   +39.976, E3 +406805.987}
SPL {X  -162.820, Y  +473.851, Z    +0.000, E1   +39.059, E3 +406818.124}
SPL {X  -162.820, Y  +470.157, Z    +0.000, E1   +38.016, E3 +406834.061}
SPL {X  -162.820, Y  +467.216, Z    +0.000, E1   +37.215, E3 +406846.823}
SPL {X  -162.820, Y  +462.598, Z    +0.000, E1   +37.325, E3 +406858.777}
SPL {X  -162.820, Y  +457.832, Z    +0.000, E1   +37.294, E3 +406872.064}
SPL {X  -162.820, Y  +452.986, Z    +0.000, E1   +37.368, E3 +406884.797}
SPL {X  -162.820, Y  +448.311, Z    +0.000, E1   +37.333, E3 +406897.817}
SPL {X  -162.820, Y  +443.351, Z    +0.000, E1   +37.335, E3 +406911.347}
SPL {X  -162.820, Y  +438.727, Z    +0.000, E1   +37.289, E3 +406924.219}
SPL {X  -162.820, Y  +434.320, Z    +0.000, E1   +37.343, E3 +406935.929}
SPL {X  -162.820, Y  +430.091, Z    +0.000, E1   +37.424, E3 +406946.929}
SPL {X  -162.820, Y  +426.177, Z    +0.000, E1   +37.250, E3 +406958.752}
SPL {X  -162.820, Y  +421.391, Z    +0.000, E1   +37.346, E3 +406971.216}
SPL {X  -162.820, Y  +416.811, Z    +0.000, E1   +37.348, E3 +406983.750}
SPL {X  -162.820, Y  +411.860, Z    +0.000, E1   +37.402, E3 +406996.902}
SPL {X  -162.820, Y  +407.726, Z    +0.000, E1   +37.291, E3 +407008.850}
SPL {X  -162.820, Y  +403.543, Z    +0.000, E1   +37.305, E3 +407020.195}
SPL {X  -162.820, Y  +399.300, Z    +0.000, E1   +37.355, E3 +407031.479}
SPL {X  -162.820, Y  +395.182, Z    +0.000, E1   +37.347, E3 +407042.768}
SPL {X  -162.820, Y  +390.797, Z    +0.000, E1   +37.358, E3 +407054.680}
SPL {X  -162.820, Y  +386.671, Z    +0.000, E1   +37.363, E3 +407065.862}
SPL {X  -162.820, Y  +382.174, Z    +0.000, E1   +37.329, E3 +407078.439}
SPL {X  -162.785, Y  +377.133, Z    +0.000, E1   +37.299, E3 +407092.368}
SPL {X  -162.576, Y  +371.586, Z    +0.000, E1   +37.322, E3 +407107.481}
SPL {X  -162.256, Y  +366.963, Z    +0.000, E1   +37.251, E3 +407120.369}
SPL {X  -161.920, Y  +363.407, Z    +0.000, E1   +37.164, E3 +407130.654}
SPL {X  -161.482, Y  +359.669, Z    +0.000, E1   +37.064, E3 +407141.439}
SPL {X  -160.943, Y  +355.851, Z    +0.000, E1   +37.136, E3 +407151.426}
SPL {X  -160.493, Y  +353.069, Z    +0.000, E1   +36.789, E3 +407161.078}
SPL {X  -159.837, Y  +349.474, Z    +0.000, E1   +36.824, E3 +407170.743}
SPL {X  -158.862, Y  +344.820, Z    +0.000, E1   +36.732, E3 +407184.106}
SPL {X  -157.959, Y  +341.011, Z    +0.000, E1   +36.448, E3 +407196.003}
SPL {X  -153.520, Y  +326.260, Z    +0.000, E1   +41.363, E3 +407204.835}
SPL {X  -150.942, Y  +319.452, Z    +0.000, E1   +36.529, E3 +407261.192}
ENDSPLINE

SPLINE
SPL {X  -159.264, Y  +346.659, Z    +0.000, E1   +22.083, E3 +407301.766}
SPL {X  -161.245, Y  +357.907, Z    +0.000, E1   +16.095, E3 +407315.199}
SPL {X  -162.697, Y  +374.161, Z    +0.000, E1    +7.119, E3 +407313.188}
SPL {X  -162.820, Y  +380.878, Z    +0.000, E1    +2.854, E3 +407316.020}
SPL {X  -162.820, Y  +385.313, Z    +0.000, E1    -0.228, E3 +407315.800}
SPL {X  -162.820, Y  +389.965, Z    +0.000, E1    -3.918, E3 +407315.168}
SPL {X  -162.820, Y  +394.532, Z    +0.000, E1    -7.849, E3 +407316.716}
SPL {X  -162.820, Y  +400.765, Z    +0.000, E1   -14.108, E3 +407314.183}
SPL {X  -162.820, Y  +411.829, Z    +0.000, E1   -24.195, E3 +407316.261}
SPL {X  -162.820, Y  +434.900, Z    +0.000, E1   -34.666, E3 +407343.625}
SPL {X  -162.820, Y  +465.440, Z    +0.000, E1   -41.264, E3 +407384.933}
ENDSPLINE

SPLINE
SPL {X  -162.820, Y  +460.175, Z    +0.000, E1   -36.098, E3 +407402.733}
ENDSPLINE

SPLINE
SPL {X  -162.820, Y  +465.690, Z    +0.000, E1   -36.140, E3 +407418.047}
SPL {X  -162.820, Y  +470.432, Z    +0.000, E1   -36.100, E3 +407431.929}
SPL {X  -162.820, Y  +475.701, Z    +0.000, E1   -36.157, E3 +407446.557}
SPL {X  -162.820, Y  +479.954, Z    +0.000, E1   -36.086, E3 +407459.097}
SPL {X  -162.820, Y  +483.976, Z    +0.000, E1   -36.049, E3 +407470.829}
SPL {X  -162.820, Y  +488.601, Z    +0.000, E1   -36.081, E3 +407483.919}
SPL {X  -162.820, Y  +493.837, Z    +0.000, E1   -36.178, E3 +407498.262}
SPL {X  -162.820, Y  +497.796, Z    +0.000, E1   -36.022, E3 +407510.447}
SPL {X  -162.820, Y  +502.146, Z    +0.000, E1   -36.123, E3 +407522.316}
SPL {X  -162.820, Y  +505.688, Z    +0.000, E1   -36.050, E3 +407532.798}
SPL {X  -162.820, Y  +509.364, Z    +0.000, E1   -36.084, E3 +407543.169}
SPL {X  -162.820, Y  +513.393, Z    +0.000, E1   -36.179, E3 +407554.025}
SPL {X  -162.820, Y  +516.436, Z    +0.000, E1   -36.094, E3 +407563.220}
SPL {X  -162.820, Y  +520.482, Z    +0.000, E1   -36.096, E3 +407574.852}
SPL {X  -162.820, Y  +524.107, Z    +0.000, E1   -36.045, E3 +407585.436}
SPL {X  -162.820, Y  +527.962, Z    +0.000, E1   -36.074, E3 +407596.369}
SPL {X  -162.820, Y  +532.253, Z    +0.000, E1   -36.170, E3 +407607.958}
SPL {X  -162.820, Y  +536.031, Z    +0.000, E1   -36.058, E3 +407619.496}
SPL {X  -162.820, Y  +541.179, Z    +0.000, E1   -36.085, E3 +407634.136}
SPL {X  -162.820, Y  +546.355, Z    +0.000, E1   -36.114, E3 +407648.681}
SPL {X  -162.820, Y  +551.776, Z    +0.000, E1   -36.108, E3 +407664.315}
SPL {X  -162.820, Y  +556.944, Z    +0.000, E1   -36.118, E3 +407678.885}
SPL {X  -162.820, Y  +561.684, Z    +0.000, E1   -36.118, E3 +407692.477}
SPL {X  -162.820, Y  +566.500, Z    +0.000, E1   -36.073, E3 +407706.480}
SPL {X  -162.820, Y  +571.734, Z    +0.000, E1   -36.094, E3 +407721.410}
SPL {X  -162.820, Y  +576.887, Z    +0.000, E1   -36.084, E3 +407736.103}
SPL {X  -162.820, Y  +581.763, Z    +0.000, E1   -36.093, E3 +407750.040}
SPL {X  -162.820, Y  +586.693, Z    +0.000, E1   -36.086, E3 +407764.145}
SPL {X  -162.820, Y  +590.250, Z    +0.000, E1   -36.075, E3 +407774.263}
SPL {X  -162.820, Y  +592.727, Z    +0.000, E1   -35.960, E3 +407782.088}
SPL {X  -162.820, Y  +597.399, Z    +0.000, E1   -36.147, E3 +407794.436}
SPL {X  -162.820, Y  +602.243, Z    +0.000, E1   -36.085, E3 +407808.582}
SPL {X  -162.820, Y  +606.975, Z    +0.000, E1   -36.102, E3 +407822.027}
SPL {X  -162.820, Y  +611.980, Z    +0.000, E1   -36.072, E3 +407836.573}
SPL {X  -162.820, Y  +616.897, Z    +0.000, E1   -36.061, E3 +407850.621}
SPL {X  -162.820, Y  +621.516, Z    +0.000, E1   -36.072, E3 +407863.820}
SPL {X  -162.820, Y  +626.243, Z    +0.000, E1   -36.105, E3 +407877.063}
SPL {X  -162.820, Y  +630.571, Z    +0.000, E1   -36.057, E3 +407889.765}
SPL {X  -162.820, Y  +634.189, Z    +0.000, E1   -36.065, E3 +407899.959}
SPL {X  -162.820, Y  +638.473, Z    +0.000, E1   -36.098, E3 +407912.196}
SPL {X  -162.820, Y  +642.832, Z    +0.000, E1   -36.091, E3 +407924.522}
SPL {X  -162.820, Y  +646.320, Z    +0.000, E1   -36.078, E3 +407934.629}
SPL {X  -162.820, Y  +649.997, Z    +0.000, E1   -36.000, E3 +407945.599}
SPL {X  -162.820, Y  +655.571, Z    +0.000, E1   -36.141, E3 +407960.934}
SPL {X  -162.820, Y  +661.560, Z    +0.000, E1   -36.068, E3 +407978.361}
SPL {X  -162.820, Y  +666.386, Z    +0.000, E1   -36.048, E3 +407992.246}
SPL {X  -162.820, Y  +672.345, Z    +0.000, E1   -36.097, E3 +408009.186}
SPL {X  -162.761, Y  +677.889, Z    +0.000, E1   -36.122, E3 +408024.651}
SPL {X  -162.577, Y  +682.401, Z    +0.000, E1   -36.021, E3 +408038.268}
SPL {X  -162.296, Y  +686.558, Z    +0.000, E1   -35.952, E3 +408050.458}
SPL {X  -161.948, Y  +690.331, Z    +0.000, E1   -35.960, E3 +408061.256}
SPL {X  -161.544, Y  +693.846, Z    +0.000, E1   -35.908, E3 +408071.531}
SPL {X  -160.925, Y  +698.267, Z    +0.000, E1   -35.816, E3 +408084.964}
SPL {X  -160.151, Y  +702.861, Z    +0.000, E1   -35.643, E3 +408098.934}
SPL {X  -159.317, Y  +707.091, Z    +0.000, E1   -35.482, E3 +408112.137}
SPL {X  -158.510, Y  +710.714, Z    +0.000, E1   -35.230, E3 +408123.848}
SPL {X  -155.037, Y  +723.239, Z    +0.000, E1   -39.382, E3 +408132.944}
SPL {X  -152.141, Y  +731.494, Z    +0.000, E1   -35.181, E3 +408191.750}
ENDSPLINE

SPLINE
SPL {X  -152.670, Y  +730.088, Z    +0.000, E1   -30.916, E3 +408265.112}
SPL {X  -160.727, Y  +699.521, Z    +0.000, E1   -18.202, E3 +408231.395}
SPL {X  -161.979, Y  +690.023, Z    +0.000, E1   -12.991, E3 +408238.205}
SPL {X  -162.641, Y  +681.139, Z    +0.000, E1    -7.893, E3 +408240.297}
SPL {X  -162.815, Y  +674.833, Z    +0.000, E1    -4.093, E3 +408237.913}
SPL {X  -162.820, Y  +669.862, Z    +0.000, E1    -0.751, E3 +408241.131}
SPL {X  -162.820, Y  +664.572, Z    +0.000, E1    +3.252, E3 +408240.945}
SPL {X  -162.820, Y  +657.781, Z    +0.000, E1    +9.391, E3 +408238.768}
SPL {X  -162.820, Y  +648.706, Z    +0.000, E1   +17.761, E3 +408240.519}
SPL {X  -162.820, Y  +635.926, Z    +0.000, E1   +28.192, E3 +408245.346}
SPL {X  -162.820, Y  +621.673, Z    +0.000, E1   +34.265, E3 +408261.704}
SPL {X  -162.820, Y  +609.002, Z    +0.000, E1   +38.458, E3 +408274.926}
SPL {X  -162.820, Y  +596.392, Z    +0.000, E1   +37.895, E3 +408308.395}
ENDSPLINE

SPLINE
SPL {X  -162.820, Y  +601.432, Z    +0.000, E1   +34.026, E3 +408317.693}
ENDSPLINE

SPLINE
SPL {X  -162.820, Y  +597.570, Z    +0.000, E1   +33.919, E3 +408330.590}
SPL {X  -162.820, Y  +592.692, Z    +0.000, E1   +33.779, E3 +408346.482}
SPL {X  -162.820, Y  +588.795, Z    +0.000, E1   +33.876, E3 +408357.919}
SPL {X  -162.820, Y  +584.646, Z    +0.000, E1   +33.882, E3 +408370.883}
SPL {X  -162.820, Y  +579.919, Z    +0.000, E1   +33.857, E3 +408385.671}
SPL {X  -162.820, Y  +574.615, Z    +0.000, E1   +33.920, E3 +408401.845}
SPL {X  -162.820, Y  +570.335, Z    +0.000, E1   +33.821, E3 +408415.550}
SPL {X  -162.820, Y  +565.901, Z    +0.000, E1   +33.889, E3 +408429.071}
SPL {X  -162.820, Y  +562.173, Z    +0.000, E1   +33.897, E3 +408440.362}
SPL {X  -162.820, Y  +559.395, Z    +0.000, E1   +33.796, E3 +408449.729}
SPL {X  -162.820, Y  +554.453, Z    +0.000, E1   +33.841, E3 +408464.954}
SPL {X  -162.820, Y  +549.726, Z    +0.000, E1   +33.905, E3 +408479.057}
SPL {X  -162.820, Y  +545.760, Z    +0.000, E1   +33.901, E3 +408491.453}
SPL {X  -162.820, Y  +541.668, Z    +0.000, E1   +33.787, E3 +408504.853}
SPL {X  -162.820, Y  +537.061, Z    +0.000, E1   +33.897, E3 +408518.511}
SPL {X  -162.820, Y  +532.164, Z    +0.000, E1   +33.861, E3 +408533.985}
SPL {X  -162.820, Y  +528.475, Z    +0.000, E1   +33.876, E3 +408545.154}
SPL {X  -162.820, Y  +524.900, Z    +0.000, E1   +33.820, E3 +408556.813}
SPL {X  -162.820, Y  +520.532, Z    +0.000, E1   +33.805, E3 +408570.380}
SPL {X  -162.820, Y  +516.814, Z    +0.000, E1   +33.917, E3 +408581.216}
SPL {X  -162.820, Y  +512.685, Z    +0.000, E1   +33.830, E3 +408594.659}
SPL {X  -162.820, Y  +508.888, Z    +0.000, E1   +33.871, E3 +408606.074}
SPL {X  -162.820, Y  +505.651, Z    +0.000, E1   +33.839, E3 +408616.391}
SPL {X  -162.820, Y  +500.931, Z    +0.000, E1   +34.256, E3 +408628.264}
SPL {X  -162.820, Y  +481.122, Z    +0.000, E1   +41.279, E3 +408638.529}
SPL {X  -162.820, Y  +478.698, Z    +0.000, E1   +40.526, E3 +408648.878}
SPL {X  -162.820, Y  +475.203, Z    +0.000, E1   +39.596, E3 +408663.337}
SPL {X  -162.820, Y  +472.097, Z    +0.000, E1   +38.411, E3 +408678.304}
SPL {X  -162.820, Y  +469.308, Z    +0.000, E1   +37.839, E3 +408689.108}
SPL {X  -162.820, Y  +467.216, Z    +0.000, E1   +37.215, E3 +408698.675}
SPL {X  -162.820, Y  +462.598, Z    +0.000, E1   +37.325, E3 +408710.629}
SPL {X  -162.820, Y  +457.832, Z    +0.000, E1   +37.294, E3 +408723.915}
SPL {X  -162.820, Y  +452.986, Z    +0.000, E1   +37.368, E3 +408736.649}
SPL {X  -162.820, Y  +448.311, Z    +0.000, E1   +37.333, E3 +408749.669}
SPL {X  -162.820, Y  +443.351, Z    +0.000, E1   +37.335, E3 +408763.199}
SPL {X  -162.820, Y  +438.727, Z    +0.000, E1   +37.289, E3 +408776.071}
SPL {X  -162.820, Y  +434.320, Z    +0.000, E1   +37.343, E3 +408787.781}
SPL {X  -162.820, Y  +430.091, Z    +0.000, E1   +37.424, E3 +408798.781}
SPL {X  -162.820, Y  +426.177, Z    +0.000, E1   +37.250, E3 +408810.604}
SPL {X  -162.820, Y  +420.241, Z    +0.000, E1   +37.355, E3 +408826.311}
SPL {X  -162.820, Y  +415.595, Z    +0.000, E1   +37.375, E3 +408838.651}
SPL {X  -162.820, Y  +411.860, Z    +0.000, E1   +37.402, E3 +408848.754}
SPL {X  -162.820, Y  +407.726, Z    +0.000, E1   +37.291, E3 +408860.701}
SPL {X  -162.820, Y  +403.543, Z    +0.000, E1   +37.305, E3 +408872.047}
SPL {X  -162.820, Y  +399.300, Z    +0.000, E1   +37.355, E3 +408883.331}
SPL {X  -162.820, Y  +395.182, Z    +0.000, E1   +37.347, E3 +408894.620}
SPL {X  -162.820, Y  +390.797, Z    +0.000, E1   +37.358, E3 +408906.532}
SPL {X  -162.820, Y  +386.671, Z    +0.000, E1   +37.363, E3 +408917.713}
SPL {X  -162.820, Y  +382.174, Z    +0.000, E1   +37.329, E3 +408930.291}
SPL {X  -162.785, Y  +377.133, Z    +0.000, E1   +37.299, E3 +408944.220}
SPL {X  -162.576, Y  +371.586, Z    +0.000, E1   +37.322, E3 +408959.333}
SPL {X  -162.256, Y  +366.963, Z    +0.000, E1   +37.251, E3 +408972.221}
SPL {X  -161.920, Y  +363.407, Z    +0.000, E1   +37.164, E3 +408982.506}
SPL {X  -161.341, Y  +358.603, Z    +0.000, E1   +37.117, E3 +408995.987}
SPL {X  -160.616, Y  +353.801, Z    +0.000, E1   +36.942, E3 +409010.151}
SPL {X  -159.837, Y  +349.474, Z    +0.000, E1   +36.824, E3 +409022.595}
SPL {X  -159.171, Y  +346.224, Z    +0.000, E1   +36.747, E3 +409031.872}
SPL {X  -158.248, Y  +342.188, Z    +0.000, E1   +36.583, E3 +409044.034}
SPL {X  -153.520, Y  +326.260, Z    +0.000, E1   +41.363, E3 +409056.687}
SPL {X  -150.942, Y  +319.452, Z    +0.000, E1   +36.529, E3 +409113.044}
ENDSPLINE

SPLINE
SPL {X  -159.264, Y  +346.659, Z    +0.000, E1   +22.083, E3 +409153.618}
SPL {X  -161.245, Y  +357.907, Z    +0.000, E1   +16.095, E3 +409167.051}
SPL {X  -162.697, Y  +374.161, Z    +0.000, E1    +7.119, E3 +409165.040}
SPL {X  -162.820, Y  +380.878, Z    +0.000, E1    +2.854, E3 +409167.872}
SPL {X  -162.820, Y  +385.313, Z    +0.000, E1    -0.228, E3 +409167.652}
SPL {X  -162.820, Y  +389.965, Z    +0.000, E1    -3.918, E3 +409167.020}
SPL {X  -162.820, Y  +394.532, Z    +0.000, E1    -7.849, E3 +409168.568}
SPL {X  -162.820, Y  +400.765, Z    +0.000, E1   -14.108, E3 +409166.035}
SPL {X  -162.820, Y  +411.829, Z    +0.000, E1   -24.195, E3 +409168.113}
SPL {X  -162.820, Y  +434.900, Z    +0.000, E1   -34.666, E3 +409195.477}
SPL {X  -162.820, Y  +465.440, Z    +0.000, E1   -41.264, E3 +409236.785}
ENDSPLINE

SPLINE
SPL {X  -162.820, Y  +460.175, Z    +0.000, E1   -36.098, E3 +409254.584}
ENDSPLINE

SPLINE
SPL {X  -162.820, Y  +465.690, Z    +0.000, E1   -36.140, E3 +409269.899}
SPL {X  -162.820, Y  +470.432, Z    +0.000, E1   -36.100, E3 +409283.781}
SPL {X  -162.820, Y  +475.701, Z    +0.000, E1   -36.157, E3 +409298.408}
SPL {X  -162.820, Y  +479.954, Z    +0.000, E1   -36.086, E3 +409310.949}
SPL {X  -162.820, Y  +485.438, Z    +0.000, E1   -36.112, E3 +409326.667}
SPL {X  -162.820, Y  +490.843, Z    +0.000, E1   -36.087, E3 +409342.080}
SPL {X  -162.820, Y  +494.712, Z    +0.000, E1   -36.164, E3 +409352.593}
SPL {X  -162.820, Y  +497.796, Z    +0.000, E1   -36.022, E3 +409362.299}
SPL {X  -162.820, Y  +502.146, Z    +0.000, E1   -36.123, E3 +409374.168}
SPL {X  -162.820, Y  +505.688, Z    +0.000, E1   -36.050, E3 +409384.650}
SPL {X  -162.820, Y  +509.364, Z    +0.000, E1   -36.084, E3 +409395.020}
SPL {X  -162.820, Y  +513.393, Z    +0.000, E1   -36.179, E3 +409405.876}
SPL {X  -162.820, Y  +516.436, Z    +0.000, E1   -36.094, E3 +409415.072}
SPL {X  -162.820, Y  +520.482, Z    +0.000, E1   -36.096, E3 +409426.704}
SPL {X  -162.820, Y  +524.107, Z    +0.000, E1   -36.045, E3 +409437.288}
SPL {X  -162.820, Y  +527.962, Z    +0.000, E1   -36.074, E3 +409448.221}
SPL {X  -162.820, Y  +532.253, Z    +0.000, E1   -36.170, E3 +409459.810}
SPL {X  -162.820, Y  +536.031, Z    +0.000, E1   -36.058, E3 +409471.348}
SPL {X  -162.820, Y  +541.179, Z    +0.000, E1   -36.085, E3 +409485.988}
SPL {X  -162.820, Y  +546.355, Z    +0.000, E1   -36.114, E3 +409500.533}
SPL {X  -162.820, Y  +551.776, Z    +0.000, E1   -36.108, E3 +409516.166}
SPL {X  -162.820, Y  +558.272, Z    +0.000, E1   -36.170, E3 +409534.375}
SPL {X  -162.820, Y  +562.721, Z    +0.000, E1   -36.046, E3 +409547.600}
SPL {X  -162.820, Y  +566.500, Z    +0.000, E1   -36.073, E3 +409558.332}
SPL {X  -162.820, Y  +570.319, Z    +0.000, E1   -36.045, E3 +409569.360}
SPL {X  -162.820, Y  +573.265, Z    +0.000, E1   -36.071, E3 +409577.597}
SPL {X  -162.820, Y  +576.887, Z    +0.000, E1   -36.084, E3 +409587.955}
SPL {X  -162.820, Y  +581.763, Z    +0.000, E1   -36.093, E3 +409601.892}
SPL {X  -162.820, Y  +586.693, Z    +0.000, E1   -36.086, E3 +409615.997}
SPL {X  -162.820, Y  +591.665, Z    +0.000, E1   -36.045, E3 +409630.524}
SPL {X  -162.820, Y  +597.399, Z    +0.000, E1   -36.147, E3 +409646.288}
SPL {X  -162.820, Y  +602.243, Z    +0.000, E1   -36.085, E3 +409660.434}
SPL {X  -162.820, Y  +605.848, Z    +0.000, E1   -36.070, E3 +409670.755}
SPL {X  -162.820, Y  +609.375, Z    +0.000, E1   -36.084, E3 +409680.805}
SPL {X  -162.820, Y  +612.959, Z    +0.000, E1   -36.034, E3 +409691.326}
SPL {X  -162.820, Y  +616.897, Z    +0.000, E1   -36.061, E3 +409702.473}
SPL {X  -162.820, Y  +621.516, Z    +0.000, E1   -36.072, E3 +409715.672}
SPL {X  -162.820, Y  +626.243, Z    +0.000, E1   -36.105, E3 +409728.915}
SPL {X  -162.820, Y  +630.571, Z    +0.000, E1   -36.057, E3 +409741.617}
SPL {X  -162.820, Y  +634.189, Z    +0.000, E1   -36.065, E3 +409751.811}
SPL {X  -162.820, Y  +638.473, Z    +0.000, E1   -36.098, E3 +409764.047}
SPL {X  -162.820, Y  +642.832, Z    +0.000, E1   -36.091, E3 +409776.373}
SPL {X  -162.820, Y  +646.320, Z    +0.000, E1   -36.078, E3 +409786.481}
SPL {X  -162.820, Y  +649.997, Z    +0.000, E1   -36.000, E3 +409797.451}
SPL {X  -162.820, Y  +655.571, Z    +0.000, E1   -36.141, E3 +409812.786}
SPL {X  -162.820, Y  +661.560, Z    +0.000, E1   -36.068, E3 +409830.213}
SPL {X  -162.820, Y  +667.641, Z    +0.000, E1   -36.092, E3 +409847.594}
SPL {X  -162.820, Y  +673.415, Z    +0.000, E1   -36.053, E3 +409864.185}
SPL {X  -162.761, Y  +677.889, Z    +0.000, E1   -36.122, E3 +409876.503}
SPL {X  -162.577, Y  +682.401, Z    +0.000, E1   -36.021, E3 +409890.119}
SPL {X  -162.187, Y  +687.846, Z    +0.000, E1   -36.007, E3 +409905.788}
SPL {X  -161.667, Y  +692.839, Z    +0.000, E1   -35.918, E3 +409920.554}
SPL {X  -161.078, Y  +697.256, Z    +0.000, E1   -35.797, E3 +409933.890}
SPL {X  -160.313, Y  +701.964, Z    +0.000, E1   -35.709, E3 +409947.965}
SPL {X  -159.317, Y  +707.091, Z    +0.000, E1   -35.482, E3 +409963.989}
SPL {X  -158.510, Y  +710.714, Z    +0.000, E1   -35.230, E3 +409975.700}
SPL {X  -155.037, Y  +723.239, Z    +0.000, E1   -39.382, E3 +409984.796}
SPL {X  -152.141, Y  +731.494, Z    +0.000, E1   -35.181, E3 +410043.602}
ENDSPLINE

SPLINE
SPL {X  -152.670, Y  +730.088, Z    +0.000, E1   -30.916, E3 +410116.964}
SPL {X  -160.727, Y  +699.521, Z    +0.000, E1   -18.202, E3 +410083.247}
SPL {X  -161.979, Y  +690.023, Z    +0.000, E1   -12.991, E3 +410090.057}
SPL {X  -162.641, Y  +681.139, Z    +0.000, E1    -7.893, E3 +410092.149}
SPL {X  -162.820, Y  +673.062, Z    +0.000, E1    -2.992, E3 +410091.116}
SPL {X  -162.820, Y  +666.731, Z    +0.000, E1    +1.545, E3 +410092.746}
SPL {X  -162.820, Y  +660.758, Z    +0.000, E1    +6.523, E3 +410092.456}
SPL {X  -162.820, Y  +650.583, Z    +0.000, E1   +16.035, E3 +410091.429}
SPL {X  -162.820, Y  +629.267, Z    +0.000, E1   +31.872, E3 +410102.577}
SPL {X  -162.820, Y  +617.390, Z    +0.000, E1   +35.413, E3 +410119.507}
SPL {X  -162.820, Y  +596.392, Z    +0.000, E1   +37.895, E3 +410160.247}
ENDSPLINE

SPLINE
SPL {X  -162.820, Y  +599.924, Z    +0.000, E1   +33.992, E3 +410174.620}
ENDSPLINE

SPLINE
SPL {X  -162.820, Y  +596.128, Z    +0.000, E1   +33.827, E3 +410187.258}
SPL {X  -162.820, Y  +592.692, Z    +0.000, E1   +33.779, E3 +410198.334}
SPL {X  -162.820, Y  +588.795, Z    +0.000, E1   +33.876, E3 +410209.771}
SPL {X  -162.820, Y  +585.519, Z    +0.000, E1   +33.888, E3 +410219.855}
SPL {X  -162.820, Y  +582.066, Z    +0.000, E1   +33.857, E3 +410230.789}
SPL {X  -162.820, Y  +577.919, Z    +0.000, E1   +33.841, E3 +410243.843}
SPL {X  -162.820, Y  +573.566, Z    +0.000, E1   +33.899, E3 +410256.918}
SPL {X  -162.820, Y  +569.298, Z    +0.000, E1   +33.851, E3 +410270.559}
SPL {X  -162.820, Y  +565.024, Z    +0.000, E1   +33.872, E3 +410283.615}
SPL {X  -162.820, Y  +560.226, Z    +0.000, E1   +33.868, E3 +410298.708}
SPL {X  -162.820, Y  +556.206, Z    +0.000, E1   +33.843, E3 +410311.108}
SPL {X  -162.820, Y  +553.486, Z    +0.000, E1   +33.777, E3 +410320.054}
SPL {X  -162.820, Y  +548.576, Z    +0.000, E1   +33.950, E3 +410334.336}
SPL {X  -162.820, Y  +544.808, Z    +0.000, E1   +33.827, E3 +410346.599}
SPL {X  -162.820, Y  +541.668, Z    +0.000, E1   +33.787, E3 +410356.705}
SPL {X  -162.820, Y  +538.174, Z    +0.000, E1   +33.865, E3 +410366.994}
SPL {X  -162.820, Y  +534.943, Z    +0.000, E1   +33.919, E3 +410376.735}
SPL {X  -162.820, Y  +531.459, Z    +0.000, E1   +33.783, E3 +410388.392}
SPL {X  -162.820, Y  +528.475, Z    +0.000, E1   +33.876, E3 +410397.006}
SPL {X  -162.820, Y  +524.900, Z    +0.000, E1   +33.820, E3 +410408.665}
SPL {X  -162.820, Y  +520.532, Z    +0.000, E1   +33.805, E3 +410422.232}
SPL {X  -162.820, Y  +515.754, Z    +0.000, E1   +33.911, E3 +410436.568}
SPL {X  -162.820, Y  +510.207, Z    +0.000, E1   +33.879, E3 +410453.949}
SPL {X  -162.820, Y  +505.651, Z    +0.000, E1   +33.839, E3 +410468.243}
SPL {X  -162.820, Y  +500.931, Z    +0.000, E1   +34.256, E3 +410480.116}
SPL {X  -162.820, Y  +481.122, Z    +0.000, E1   +41.279, E3 +410490.381}
SPL {X  -162.820, Y  +478.698, Z    +0.000, E1   +40.526, E3 +410500.730}
SPL {X  -162.820, Y  +475.203, Z    +0.000, E1   +39.596, E3 +410515.189}
SPL {X  -162.820, Y  +472.097, Z    +0.000, E1   +38.411, E3 +410530.156}
SPL {X  -162.820, Y  +469.308, Z    +0.000, E1   +37.839, E3 +410540.960}
SPL {X  -162.820, Y  +467.216, Z    +0.000, E1   +37.215, E3 +410550.527}
SPL {X  -162.820, Y  +462.598, Z    +0.000, E1   +37.325, E3 +410562.481}
SPL {X  -162.820, Y  +457.832, Z    +0.000, E1   +37.294, E3 +410575.767}
SPL {X  -162.820, Y  +452.986, Z    +0.000, E1   +37.368, E3 +410588.501}
SPL {X  -162.820, Y  +448.311, Z    +0.000, E1   +37.333, E3 +410601.521}
SPL {X  -162.820, Y  +443.351, Z    +0.000, E1   +37.335, E3 +410615.051}
SPL {X  -162.820, Y  +438.727, Z    +0.000, E1   +37.289, E3 +410627.923}
SPL {X  -162.820, Y  +434.320, Z    +0.000, E1   +37.343, E3 +410639.633}
SPL {X  -162.820, Y  +430.091, Z    +0.000, E1   +37.424, E3 +410650.633}
SPL {X  -162.820, Y  +426.177, Z    +0.000, E1   +37.250, E3 +410662.456}
SPL {X  -162.820, Y  +421.391, Z    +0.000, E1   +37.346, E3 +410674.920}
SPL {X  -162.820, Y  +416.811, Z    +0.000, E1   +37.348, E3 +410687.454}
SPL {X  -162.820, Y  +411.860, Z    +0.000, E1   +37.402, E3 +410700.605}
SPL {X  -162.820, Y  +407.726, Z    +0.000, E1   +37.291, E3 +410712.553}
SPL {X  -162.820, Y  +403.543, Z    +0.000, E1   +37.305, E3 +410723.899}
SPL {X  -162.820, Y  +399.300, Z    +0.000, E1   +37.355, E3 +410735.183}
SPL {X  -162.820, Y  +395.182, Z    +0.000, E1   +37.347, E3 +410746.472}
SPL {X  -162.820, Y  +390.797, Z    +0.000, E1   +37.358, E3 +410758.384}
SPL {X  -162.820, Y  +386.671, Z    +0.000, E1   +37.363, E3 +410769.565}
SPL {X  -162.820, Y  +382.174, Z    +0.000, E1   +37.329, E3 +410782.143}
SPL {X  -162.785, Y  +377.133, Z    +0.000, E1   +37.299, E3 +410796.072}
SPL {X  -162.623, Y  +372.484, Z    +0.000, E1   +37.337, E3 +410808.511}
SPL {X  -162.331, Y  +367.894, Z    +0.000, E1   +37.251, E3 +410821.624}
SPL {X  -161.920, Y  +363.407, Z    +0.000, E1   +37.164, E3 +410834.358}
SPL {X  -161.482, Y  +359.669, Z    +0.000, E1   +37.064, E3 +410845.143}
SPL {X  -160.943, Y  +355.851, Z    +0.000, E1   +37.136, E3 +410855.129}
SPL {X  -160.493, Y  +353.069, Z    +0.000, E1   +36.789, E3 +410864.781}
SPL {X  -159.837, Y  +349.474, Z    +0.000, E1   +36.824, E3 +410874.447}
SPL {X  -158.862, Y  +344.820, Z    +0.000, E1   +36.732, E3 +410887.809}
SPL {X  -157.959, Y  +341.011, Z    +0.000, E1   +36.448, E3 +410899.706}
SPL {X  -154.495, Y  +329.104, Z    +0.000, E1   +40.891, E3 +410904.589}
SPL {X  -152.543, Y  +323.569, Z    +0.000, E1   +41.772, E3 +410912.345}
SPL {X  -150.942, Y  +319.452, Z    +0.000, E1   +36.529, E3 +410964.896}
ENDSPLINE

SPLINE
SPL {X  -160.206, Y  +351.441, Z    +0.000, E1   +19.697, E3 +411009.266}
SPL {X  -161.531, Y  +360.055, Z    +0.000, E1   +14.747, E3 +411026.152}
SPL {X  -162.746, Y  +375.590, Z    +0.000, E1    +6.280, E3 +411018.491}
SPL {X  -162.820, Y  +384.478, Z    +0.000, E1    +0.434, E3 +411019.160}
SPL {X  -162.820, Y  +389.965, Z    +0.000, E1    -3.918, E3 +411018.872}
SPL {X  -162.820, Y  +394.532, Z    +0.000, E1    -7.849, E3 +411020.420}
SPL {X  -162.820, Y  +400.765, Z    +0.000, E1   -14.108, E3 +411017.887}
SPL {X  -162.820, Y  +411.829, Z    +0.000, E1   -24.195, E3 +411019.964}
SPL {X  -162.820, Y  +434.900, Z    +0.000, E1   -34.666, E3 +411047.329}
SPL {X  -162.820, Y  +465.440, Z    +0.000, E1   -41.264, E3 +411088.637}
ENDSPLINE

SPLINE
SPL {X  -162.820, Y  +458.794, Z    +0.000, E1   -36.100, E3 +411102.260}
ENDSPLINE

SPLINE
SPL {X  -162.820, Y  +461.779, Z    +0.000, E1   -35.988, E3 +411111.456}
SPL {X  -162.820, Y  +465.690, Z    +0.000, E1   -36.140, E3 +411121.751}
SPL {X  -162.820, Y  +470.432, Z    +0.000, E1   -36.100, E3 +411135.633}
SPL {X  -162.820, Y  +475.701, Z    +0.000, E1   -36.157, E3 +411150.260}
SPL {X  -162.820, Y  +479.954, Z    +0.000, E1   -36.086, E3 +411162.801}
SPL {X  -162.820, Y  +485.438, Z    +0.000, E1   -36.112, E3 +411178.519}
SPL {X  -162.820, Y  +490.843, Z    +0.000, E1   -36.087, E3 +411193.932}
SPL {X  -162.820, Y  +494.712, Z    +0.000, E1   -36.164, E3 +411204.444}
SPL {X  -162.820, Y  +497.796, Z    +0.000, E1   -36.022, E3 +411214.151}
SPL {X  -162.820, Y  +502.146, Z    +0.000, E1   -36.123, E3 +411226.020}
SPL {X  -162.820, Y  +505.688, Z    +0.000, E1   -36.050, E3 +411236.502}
SPL {X  -162.820, Y  +509.364, Z    +0.000, E1   -36.084, E3 +411246.872}
SPL {X  -162.820, Y  +515.001, Z    +0.000, E1   -36.183, E3 +411262.510}
SPL {X  -162.820, Y  +520.482, Z    +0.000, E1   -36.096, E3 +411278.556}
SPL {X  -162.820, Y  +524.107, Z    +0.000, E1   -36.045, E3 +411289.139}
SPL {X  -162.820, Y  +527.962, Z    +0.000, E1   -36.074, E3 +411300.072}
SPL {X  -162.820, Y  +532.253, Z    +0.000, E1   -36.170, E3 +411311.661}
SPL {X  -162.820, Y  +536.031, Z    +0.000, E1   -36.058, E3 +411323.199}
SPL {X  -162.820, Y  +541.179, Z    +0.000, E1   -36.085, E3 +411337.840}
SPL {X  -162.820, Y  +546.355, Z    +0.000, E1   -36.114, E3 +411352.384}
SPL {X  -162.820, Y  +550.585, Z    +0.000, E1   -36.077, E3 +411364.654}
SPL {X  -162.820, Y  +555.903, Z    +0.000, E1   -36.136, E3 +411379.652}
SPL {X  -162.820, Y  +561.684, Z    +0.000, E1   -36.118, E3 +411396.181}
SPL {X  -162.820, Y  +566.500, Z    +0.000, E1   -36.073, E3 +411410.184}
SPL {X  -162.820, Y  +570.319, Z    +0.000, E1   -36.045, E3 +411421.212}
SPL {X  -162.820, Y  +573.265, Z    +0.000, E1   -36.071, E3 +411429.448}
SPL {X  -162.820, Y  +576.887, Z    +0.000, E1   -36.084, E3 +411439.807}
SPL {X  -162.820, Y  +581.763, Z    +0.000, E1   -36.093, E3 +411453.744}
SPL {X  -162.820, Y  +586.693, Z    +0.000, E1   -36.086, E3 +411467.848}
SPL {X  -162.820, Y  +590.250, Z    +0.000, E1   -36.075, E3 +411477.967}
SPL {X  -162.820, Y  +594.470, Z    +0.000, E1   -36.080, E3 +411490.198}
SPL {X  -162.820, Y  +598.788, Z    +0.000, E1   -36.102, E3 +411502.219}
SPL {X  -162.820, Y  +602.243, Z    +0.000, E1   -36.085, E3 +411512.286}
SPL {X  -162.820, Y  +605.848, Z    +0.000, E1   -36.070, E3 +411522.607}
SPL {X  -162.820, Y  +609.375, Z    +0.000, E1   -36.084, E3 +411532.657}
SPL {X  -162.820, Y  +612.959, Z    +0.000, E1   -36.034, E3 +411543.178}
SPL {X  -162.820, Y  +616.897, Z    +0.000, E1   -36.061, E3 +411554.325}
SPL {X  -162.820, Y  +621.516, Z    +0.000, E1   -36.072, E3 +411567.524}
SPL {X  -162.820, Y  +626.243, Z    +0.000, E1   -36.105, E3 +411580.767}
SPL {X  -162.820, Y  +630.571, Z    +0.000, E1   -36.057, E3 +411593.469}
SPL {X  -162.820, Y  +635.505, Z    +0.000, E1   -36.079, E3 +411607.475}
SPL {X  -162.820, Y  +641.277, Z    +0.000, E1   -36.126, E3 +411623.767}
SPL {X  -162.820, Y  +646.320, Z    +0.000, E1   -36.078, E3 +411638.333}
SPL {X  -162.820, Y  +651.289, Z    +0.000, E1   -36.059, E3 +411652.789}
SPL {X  -162.820, Y  +656.677, Z    +0.000, E1   -36.110, E3 +411667.802}
SPL {X  -162.820, Y  +661.560, Z    +0.000, E1   -36.068, E3 +411682.065}
SPL {X  -162.820, Y  +666.386, Z    +0.000, E1   -36.048, E3 +411695.949}
SPL {X  -162.820, Y  +672.345, Z    +0.000, E1   -36.097, E3 +411712.890}
SPL {X  -162.761, Y  +677.889, Z    +0.000, E1   -36.122, E3 +411728.355}
SPL {X  -162.577, Y  +682.401, Z    +0.000, E1   -36.021, E3 +411741.971}
SPL {X  -162.187, Y  +687.846, Z    +0.000, E1   -36.007, E3 +411757.640}
SPL {X  -161.667, Y  +692.839, Z    +0.000, E1   -35.918, E3 +411772.406}
SPL {X  -160.925, Y  +698.267, Z    +0.000, E1   -35.816, E3 +411788.667}
SPL {X  -160.151, Y  +702.861, Z    +0.000, E1   -35.643, E3 +411802.637}
SPL {X  -159.317, Y  +707.091, Z    +0.000, E1   -35.482, E3 +411815.841}
SPL {X  -158.510, Y  +710.714, Z    +0.000, E1   -35.230, E3 +411827.552}
SPL {X  -155.037, Y  +723.239, Z    +0.000, E1   -39.382, E3 +411836.648}
SPL {X  -152.141, Y  +731.494, Z    +0.000, E1   -35.181, E3 +411895.454}
ENDSPLINE

SPLINE
SPL {X  -160.133, Y  +702.956, Z    +0.000, E1   -19.806, E3 +411938.992}
SPL {X  -161.979, Y  +690.023, Z    +0.000, E1   -12.991, E3 +411941.909}
SPL {X  -162.641, Y  +681.139, Z    +0.000, E1    -7.893, E3 +411944.001}
SPL {X  -162.820, Y  +673.062, Z    +0.000, E1    -2.992, E3 +411942.967}
SPL {X  -162.820, Y  +666.731, Z    +0.000, E1    +1.545, E3 +411944.597}
SPL {X  -162.820, Y  +660.758, Z    +0.000, E1    +6.523, E3 +411944.308}
SPL {X  -162.820, Y  +650.583, Z    +0.000, E1   +16.035, E3 +411943.280}
SPL {X  -162.820, Y  +629.267, Z    +0.000, E1   +31.872, E3 +411954.429}
SPL {X  -162.820, Y  +620.680, Z    +0.000, E1   +34.107, E3 +411968.478}
SPL {X  -162.820, Y  +601.185, Z    +0.000, E1   +39.430, E3 +411991.986}
SPL {X  -162.820, Y  +599.927, Z    +0.000, E1   +35.241, E3 +412018.564}
SPL {X  -162.820, Y  +597.570, Z    +0.000, E1   +33.919, E3 +412034.294}
SPL {X  -162.820, Y  +592.692, Z    +0.000, E1   +33.779, E3 +412050.186}
SPL {X  -162.820, Y  +588.795, Z    +0.000, E1   +33.876, E3 +412061.623}
SPL {X  -162.820, Y  +585.519, Z    +0.000, E1   +33.888, E3 +412071.707}
SPL {X  -162.820, Y  +582.066, Z    +0.000, E1   +33.857, E3 +412082.641}
SPL {X  -162.820, Y  +577.919, Z    +0.000, E1   +33.841, E3 +412095.695}
SPL {X  -162.820, Y  +573.566, Z    +0.000, E1   +33.899, E3 +412108.770}
SPL {X  -162.820, Y  +569.298, Z    +0.000, E1   +33.851, E3 +412122.411}
SPL {X  -162.820, Y  +563.983, Z    +0.000, E1   +33.916, E3 +412138.551}
SPL {X  -162.820, Y  +559.395, Z    +0.000, E1   +33.796, E3 +412153.433}
SPL {X  -162.820, Y  +554.453, Z    +0.000, E1   +33.841, E3 +412168.657}
SPL {X  -162.820, Y  +549.726, Z    +0.000, E1   +33.905, E3 +412182.761}
SPL {X  -162.820, Y  +545.760, Z    +0.000, E1   +33.901, E3 +412195.157}
SPL {X  -162.820, Y  +541.668, Z    +0.000, E1   +33.787, E3 +412208.557}
SPL {X  -162.820, Y  +537.061, Z    +0.000, E1   +33.897, E3 +412222.215}
SPL {X  -162.820, Y  +532.164, Z    +0.000, E1   +33.861, E3 +412237.689}
SPL {X  -162.820, Y  +528.475, Z    +0.000, E1   +33.876, E3 +412248.858}
SPL {X  -162.820, Y  +524.900, Z    +0.000, E1   +33.820, E3 +412260.516}
SPL {X  -162.820, Y  +520.532, Z    +0.000, E1   +33.805, E3 +412274.084}
SPL {X  -162.820, Y  +516.814, Z    +0.000, E1   +33.917, E3 +412284.920}
SPL {X  -162.820, Y  +512.685, Z    +0.000, E1   +33.830, E3 +412298.363}
SPL {X  -162.820, Y  +508.888, Z    +0.000, E1   +33.871, E3 +412309.778}
SPL {X  -162.820, Y  +505.651, Z    +0.000, E1   +33.839, E3 +412320.095}
SPL {X  -162.820, Y  +500.931, Z    +0.000, E1   +34.256, E3 +412331.968}
SPL {X  -162.820, Y  +481.122, Z    +0.000, E1   +41.279, E3 +412342.233}
SPL {X  -162.820, Y  +477.698, Z    +0.000, E1   +40.353, E3 +412356.289}
SPL {X  -162.820, Y  +474.538, Z    +0.000, E1   +39.267, E3 +412370.464}
SPL {X  -162.820, Y  +472.097, Z    +0.000, E1   +38.411, E3 +412382.008}
SPL {X  -162.820, Y  +469.308, Z    +0.000, E1   +37.839, E3 +412392.812}
SPL {X  -162.820, Y  +467.216, Z    +0.000, E1   +37.215, E3 +412402.378}
SPL {X  -162.820, Y  +462.598, Z    +0.000, E1   +37.325, E3 +412414.332}
SPL {X  -162.820, Y  +457.832, Z    +0.000, E1   +37.294, E3 +412427.619}
SPL {X  -162.820, Y  +452.986, Z    +0.000, E1   +37.368, E3 +412440.353}
SPL {X  -162.820, Y  +448.311, Z    +0.000, E1   +37.333, E3 +412453.373}
SPL {X  -162.820, Y  +443.351, Z    +0.000, E1   +37.335, E3 +412466.903}
SPL {X  -162.820, Y  +438.727, Z    +0.000, E1   +37.289, E3 +412479.775}
SPL {X  -162.820, Y  +434.320, Z    +0.000, E1   +37.343, E3 +412491.485}
SPL {X  -162.820, Y  +430.091, Z    +0.000, E1   +37.424, E3 +412502.485}
SPL {X  -162.820, Y  +426.177, Z    +0.000, E1   +37.250, E3 +412514.308}
SPL {X  -162.820, Y  +421.391, Z    +0.000, E1   +37.346, E3 +412526.771}
SPL {X  -162.820, Y  +416.811, Z    +0.000, E1   +37.348, E3 +412539.306}
SPL {X  -162.820, Y  +411.860, Z    +0.000, E1   +37.402, E3 +412552.457}
SPL {X  -162.820, Y  +407.726, Z    +0.000, E1   +37.291, E3 +412564.405}
SPL {X  -162.820, Y  +403.543, Z    +0.000, E1   +37.305, E3 +412575.751}
SPL {X  -162.820, Y  +399.300, Z    +0.000, E1   +37.355, E3 +412587.035}
SPL {X  -162.820, Y  +395.182, Z    +0.000, E1   +37.347, E3 +412598.324}
SPL {X  -162.820, Y  +390.797, Z    +0.000, E1   +37.358, E3 +412610.236}
SPL {X  -162.820, Y  +386.671, Z    +0.000, E1   +37.363, E3 +412621.417}
SPL {X  -162.820, Y  +382.174, Z    +0.000, E1   +37.329, E3 +412633.995}
SPL {X  -162.785, Y  +377.133, Z    +0.000, E1   +37.299, E3 +412647.924}
SPL {X  -162.576, Y  +371.586, Z    +0.000, E1   +37.322, E3 +412663.036}
SPL {X  -162.256, Y  +366.963, Z    +0.000, E1   +37.251, E3 +412675.925}
SPL {X  -161.920, Y  +363.407, Z    +0.000, E1   +37.164, E3 +412686.210}
SPL {X  -161.341, Y  +358.603, Z    +0.000, E1   +37.117, E3 +412699.690}
SPL {X  -160.616, Y  +353.801, Z    +0.000, E1   +36.942, E3 +412713.855}
SPL {X  -159.837, Y  +349.474, Z    +0.000, E1   +36.824, E3 +412726.299}
SPL {X  -158.862, Y  +344.820, Z    +0.000, E1   +36.732, E3 +412739.661}
SPL {X  -157.959, Y  +341.011, Z    +0.000, E1   +36.448, E3 +412751.558}
SPL {X  -153.520, Y  +326.260, Z    +0.000, E1   +41.363, E3 +412760.390}
SPL {X  -150.942, Y  +319.452, Z    +0.000, E1   +36.529, E3 +412816.747}
ENDSPLINE

SPLINE
SPL {X  -159.264, Y  +346.659, Z    +0.000, E1   +22.083, E3 +412857.322}
SPL {X  -161.245, Y  +357.907, Z    +0.000, E1   +16.095, E3 +412870.754}
SPL {X  -162.697, Y  +374.161, Z    +0.000, E1    +7.119, E3 +412868.744}
SPL {X  -162.820, Y  +380.878, Z    +0.000, E1    +2.854, E3 +412871.575}
SPL {X  -162.820, Y  +385.313, Z    +0.000, E1    -0.228, E3 +412871.355}
SPL {X  -162.820, Y  +389.965, Z    +0.000, E1    -3.918, E3 +412870.724}
SPL {X  -162.820, Y  +394.532, Z    +0.000, E1    -7.849, E3 +412872.272}
SPL {X  -162.820, Y  +400.765, Z    +0.000, E1   -14.108, E3 +412869.739}
SPL {X  -162.820, Y  +411.829, Z    +0.000, E1   -24.195, E3 +412871.816}
SPL {X  -162.820, Y  +434.900, Z    +0.000, E1   -34.666, E3 +412899.181}
SPL {X  -162.820, Y  +465.440, Z    +0.000, E1   -41.264, E3 +412940.488}
ENDSPLINE

SPLINE
SPL {X  -162.820, Y  +460.175, Z    +0.000, E1   -36.098, E3 +412958.288}
ENDSPLINE

SPLINE
SPL {X  -162.820, Y  +465.690, Z    +0.000, E1   -36.140, E3 +412973.602}
SPL {X  -162.820, Y  +470.432, Z    +0.000, E1   -36.100, E3 +412987.485}
SPL {X  -162.820, Y  +475.701, Z    +0.000, E1   -36.157, E3 +413002.112}
SPL {X  -162.820, Y  +479.954, Z    +0.000, E1   -36.086, E3 +413014.653}
SPL {X  -162.820, Y  +485.438, Z    +0.000, E1   -36.112, E3 +413030.371}
SPL {X  -162.820, Y  +490.843, Z    +0.000, E1   -36.087, E3 +413045.784}
SPL {X  -162.820, Y  +494.712, Z    +0.000, E1   -36.164, E3 +413056.296}
SPL {X  -162.820, Y  +498.932, Z    +0.000, E1   -36.079, E3 +413069.023}
SPL {X  -162.820, Y  +504.528, Z    +0.000, E1   -36.109, E3 +413084.819}
SPL {X  -162.820, Y  +509.364, Z    +0.000, E1   -36.084, E3 +413098.724}
SPL {X  -162.820, Y  +515.001, Z    +0.000, E1   -36.183, E3 +413114.362}
SPL {X  -162.820, Y  +520.482, Z    +0.000, E1   -36.096, E3 +413130.407}
SPL {X  -162.820, Y  +524.107, Z    +0.000, E1   -36.045, E3 +413140.991}
SPL {X  -162.820, Y  +527.962, Z    +0.000, E1   -36.074, E3 +413151.924}
SPL {X  -162.820, Y  +532.253, Z    +0.000, E1   -36.170, E3 +413163.513}
SPL {X  -162.820, Y  +536.031, Z    +0.000, E1   -36.058, E3 +413175.051}
SPL {X  -162.820, Y  +541.179, Z    +0.000, E1   -36.085, E3 +413189.692}
SPL {X  -162.820, Y  +546.355, Z    +0.000, E1   -36.114, E3 +413204.236}
SPL {X  -162.820, Y  +551.776, Z    +0.000, E1   -36.108, E3 +413219.870}
SPL {X  -162.820, Y  +556.944, Z    +0.000, E1   -36.118, E3 +413234.441}
SPL {X  -162.820, Y  +561.684, Z    +0.000, E1   -36.118, E3 +413248.033}
SPL {X  -162.820, Y  +566.500, Z    +0.000, E1   -36.073, E3 +413262.036}
SPL {X  -162.820, Y  +570.319, Z    +0.000, E1   -36.045, E3 +413273.064}
SPL {X  -162.820, Y  +573.265, Z    +0.000, E1   -36.071, E3 +413281.300}
SPL {X  -162.820, Y  +578.070, Z    +0.000, E1   -36.120, E3 +413294.982}
SPL {X  -162.820, Y  +582.838, Z    +0.000, E1   -36.064, E3 +413308.725}
SPL {X  -162.820, Y  +586.693, Z    +0.000, E1   -36.086, E3 +413319.700}
SPL {X  -162.820, Y  +591.665, Z    +0.000, E1   -36.045, E3 +413334.228}
SPL {X  -162.820, Y  +596.059, Z    +0.000, E1   -36.124, E3 +413346.160}
SPL {X  -162.820, Y  +598.788, Z    +0.000, E1   -36.102, E3 +413354.071}
SPL {X  -162.820, Y  +602.243, Z    +0.000, E1   -36.085, E3 +413364.138}
SPL {X  -162.820, Y  +605.848, Z    +0.000, E1   -36.070, E3 +413374.459}
SPL {X  -162.820, Y  +609.375, Z    +0.000, E1   -36.084, E3 +413384.509}
SPL {X  -162.820, Y  +612.959, Z    +0.000, E1   -36.034, E3 +413395.029}
SPL {X  -162.820, Y  +616.897, Z    +0.000, E1   -36.061, E3 +413406.177}
SPL {X  -162.820, Y  +621.516, Z    +0.000, E1   -36.072, E3 +413419.376}
SPL {X  -162.820, Y  +626.243, Z    +0.000, E1   -36.105, E3 +413432.619}
SPL {X  -162.820, Y  +630.571, Z    +0.000, E1   -36.057, E3 +413445.321}
SPL {X  -162.820, Y  +635.505, Z    +0.000, E1   -36.079, E3 +413459.327}
SPL {X  -162.820, Y  +639.747, Z    +0.000, E1   -36.079, E3 +413471.353}
SPL {X  -162.820, Y  +642.832, Z    +0.000, E1   -36.091, E3 +413480.077}
SPL {X  -162.820, Y  +646.320, Z    +0.000, E1   -36.078, E3 +413490.184}
SPL {X  -162.820, Y  +649.997, Z    +0.000, E1   -36.000, E3 +413501.155}
SPL {X  -162.820, Y  +655.571, Z    +0.000, E1   -36.141, E3 +413516.489}
SPL {X  -162.820, Y  +661.560, Z    +0.000, E1   -36.068, E3 +413533.917}
SPL {X  -162.820, Y  +666.386, Z    +0.000, E1   -36.048, E3 +413547.801}
SPL {X  -162.820, Y  +672.345, Z    +0.000, E1   -36.097, E3 +413564.742}
SPL {X  -162.761, Y  +677.889, Z    +0.000, E1   -36.122, E3 +413580.206}
SPL {X  -162.577, Y  +682.401, Z    +0.000, E1   -36.021, E3 +413593.823}
SPL {X  -162.296, Y  +686.558, Z    +0.000, E1   -35.952, E3 +413606.014}
SPL {X  -161.948, Y  +690.331, Z    +0.000, E1   -35.960, E3 +413616.812}
SPL {X  -161.544, Y  +693.846, Z    +0.000, E1   -35.908, E3 +413627.087}
SPL {X  -160.925, Y  +698.267, Z    +0.000, E1   -35.816, E3 +413640.519}
SPL {X  -160.151, Y  +702.861, Z    +0.000, E1   -35.643, E3 +413654.489}
SPL {X  -159.317, Y  +707.091, Z    +0.000, E1   -35.482, E3 +413667.693}
SPL {X  -158.510, Y  +710.714, Z    +0.000, E1   -35.230, E3 +413679.404}
SPL {X  -155.037, Y  +723.239, Z    +0.000, E1   -39.382, E3 +413688.500}
SPL {X  -152.141, Y  +731.494, Z    +0.000, E1   -35.181, E3 +413747.306}
ENDSPLINE

SPLINE
SPL {X  -160.133, Y  +702.956, Z    +0.000, E1   -19.806, E3 +413790.844}
SPL {X  -161.979, Y  +690.023, Z    +0.000, E1   -12.991, E3 +413793.761}
SPL {X  -162.641, Y  +681.139, Z    +0.000, E1    -7.893, E3 +413795.852}
SPL {X  -162.820, Y  +673.062, Z    +0.000, E1    -2.992, E3 +413794.819}
SPL {X  -162.820, Y  +665.516, Z    +0.000, E1    +2.410, E3 +413796.659}
SPL {X  -162.820, Y  +657.781, Z    +0.000, E1    +9.391, E3 +413794.323}
SPL {X  -162.820, Y  +648.706, Z    +0.000, E1   +17.761, E3 +413796.075}
SPL {X  -162.820, Y  +635.926, Z    +0.000, E1   +28.192, E3 +413800.902}
SPL {X  -162.820, Y  +621.673, Z    +0.000, E1   +34.265, E3 +413817.260}
SPL {X  -162.820, Y  +609.002, Z    +0.000, E1   +38.458, E3 +413830.481}
SPL {X  -162.820, Y  +596.392, Z    +0.000, E1   +37.895, E3 +413863.950}
ENDSPLINE

SPLINE
SPL {X  -162.820, Y  +601.432, Z    +0.000, E1   +34.026, E3 +413873.248}
ENDSPLINE

SPLINE
SPL {X  -162.820, Y  +599.021, Z    +0.000, E1   +33.912, E3 +413881.466}
SPL {X  -162.820, Y  +595.170, Z    +0.000, E1   +33.784, E3 +413894.372}
SPL {X  -162.820, Y  +589.785, Z    +0.000, E1   +33.904, E3 +413910.369}
SPL {X  -162.820, Y  +585.519, Z    +0.000, E1   +33.888, E3 +413923.559}
SPL {X  -162.820, Y  +582.066, Z    +0.000, E1   +33.857, E3 +413934.493}
SPL {X  -162.820, Y  +577.919, Z    +0.000, E1   +33.841, E3 +413947.546}
SPL {X  -162.820, Y  +573.566, Z    +0.000, E1   +33.899, E3 +413960.621}
SPL {X  -162.820, Y  +570.335, Z    +0.000, E1   +33.821, E3 +413971.106}
SPL {X  -162.820, Y  +565.901, Z    +0.000, E1   +33.889, E3 +413984.626}
SPL {X  -162.820, Y  +562.173, Z    +0.000, E1   +33.897, E3 +413995.917}
SPL {X  -162.820, Y  +559.395, Z    +0.000, E1   +33.796, E3 +414005.285}
SPL {X  -162.820, Y  +554.453, Z    +0.000, E1   +33.841, E3 +414020.509}
SPL {X  -162.820, Y  +549.726, Z    +0.000, E1   +33.905, E3 +414034.613}
SPL {X  -162.820, Y  +545.760, Z    +0.000, E1   +33.901, E3 +414047.009}
SPL {X  -162.820, Y  +541.668, Z    +0.000, E1   +33.787, E3 +414060.409}
SPL {X  -162.820, Y  +538.174, Z    +0.000, E1   +33.865, E3 +414070.698}
SPL {X  -162.820, Y  +534.943, Z    +0.000, E1   +33.919, E3 +414080.438}
SPL {X  -162.820, Y  +531.459, Z    +0.000, E1   +33.783, E3 +414092.095}
SPL {X  -162.820, Y  +526.783, Z    +0.000, E1   +33.870, E3 +414106.223}
SPL {X  -162.820, Y  +521.520, Z    +0.000, E1   +33.826, E3 +414122.870}
SPL {X  -162.820, Y  +515.754, Z    +0.000, E1   +33.911, E3 +414140.272}
SPL {X  -162.820, Y  +510.207, Z    +0.000, E1   +33.879, E3 +414157.652}
SPL {X  -162.820, Y  +504.570, Z    +0.000, E1   +33.876, E3 +414175.232}
SPL {X  -162.820, Y  +498.875, Z    +0.000, E1   +34.747, E3 +414186.933}
SPL {X  -162.820, Y  +481.122, Z    +0.000, E1   +41.279, E3 +414194.084}
SPL {X  -162.820, Y  +477.698, Z    +0.000, E1   +40.353, E3 +414208.140}
SPL {X  -162.820, Y  +473.851, Z    +0.000, E1   +39.059, E3 +414225.532}
SPL {X  -162.820, Y  +470.157, Z    +0.000, E1   +38.016, E3 +414241.469}
SPL {X  -162.820, Y  +467.216, Z    +0.000, E1   +37.215, E3 +414254.230}
SPL {X  -162.820, Y  +462.598, Z    +0.000, E1   +37.325, E3 +414266.184}
SPL {X  -162.820, Y  +457.832, Z    +0.000, E1   +37.294, E3 +414279.471}
SPL {X  -162.820, Y  +452.986, Z    +0.000, E1   +37.368, E3 +414292.205}
SPL {X  -162.820, Y  +448.311, Z    +0.000, E1   +37.333, E3 +414305.225}
SPL {X  -162.820, Y  +443.351, Z    +0.000, E1   +37.335, E3 +414318.754}
SPL {X  -162.820, Y  +438.727, Z    +0.000, E1   +37.289, E3 +414331.627}
SPL {X  -162.820, Y  +434.320, Z    +0.000, E1   +37.343, E3 +414343.337}
SPL {X  -162.820, Y  +430.091, Z    +0.000, E1   +37.424, E3 +414354.337}
SPL {X  -162.820, Y  +426.177, Z    +0.000, E1   +37.250, E3 +414366.160}
SPL {X  -162.820, Y  +421.391, Z    +0.000, E1   +37.346, E3 +414378.623}
SPL {X  -162.820, Y  +416.811, Z    +0.000, E1   +37.348, E3 +414391.158}
SPL {X  -162.820, Y  +411.860, Z    +0.000, E1   +37.402, E3 +414404.309}
SPL {X  -162.820, Y  +407.726, Z    +0.000, E1   +37.291, E3 +414416.257}
SPL {X  -162.820, Y  +403.543, Z    +0.000, E1   +37.305, E3 +414427.602}
SPL {X  -162.820, Y  +399.300, Z    +0.000, E1   +37.355, E3 +414438.887}
SPL {X  -162.820, Y  +395.182, Z    +0.000, E1   +37.347, E3 +414450.176}
SPL {X  -162.820, Y  +390.797, Z    +0.000, E1   +37.358, E3 +414462.088}
SPL {X  -162.820, Y  +385.307, Z    +0.000, E1   +37.364, E3 +414477.168}
SPL {X  -162.820, Y  +380.796, Z    +0.000, E1   +37.334, E3 +414489.454}
SPL {X  -162.785, Y  +377.133, Z    +0.000, E1   +37.299, E3 +414499.776}
SPL {X  -162.576, Y  +371.586, Z    +0.000, E1   +37.322, E3 +414514.888}
SPL {X  -162.256, Y  +366.963, Z    +0.000, E1   +37.251, E3 +414527.777}
SPL {X  -161.920, Y  +363.407, Z    +0.000, E1   +37.164, E3 +414538.062}
SPL {X  -161.482, Y  +359.669, Z    +0.000, E1   +37.064, E3 +414548.847}
SPL {X  -160.943, Y  +355.851, Z    +0.000, E1   +37.136, E3 +414558.833}
SPL {X  -160.493, Y  +353.069, Z    +0.000, E1   +36.789, E3 +414568.485}
SPL {X  -159.837, Y  +349.474, Z    +0.000, E1   +36.824, E3 +414578.151}
SPL {X  -158.862, Y  +344.820, Z    +0.000, E1   +36.732, E3 +414591.513}
SPL {X  -157.959, Y  +341.011, Z    +0.000, E1   +36.448, E3 +414603.410}
SPL {X  -153.520, Y  +326.260, Z    +0.000, E1   +41.363, E3 +414612.242}
SPL {X  -150.942, Y  +319.452, Z    +0.000, E1   +36.529, E3 +414668.599}
ENDSPLINE

SPLINE
SPL {X  -159.264, Y  +346.659, Z    +0.000, E1   +22.083, E3 +414709.173}
SPL {X  -161.245, Y  +357.907, Z    +0.000, E1   +16.095, E3 +414722.606}
SPL {X  -162.697, Y  +374.161, Z    +0.000, E1    +7.119, E3 +414720.596}
SPL {X  -162.820, Y  +380.878, Z    +0.000, E1    +2.854, E3 +414723.427}
SPL {X  -162.820, Y  +385.313, Z    +0.000, E1    -0.228, E3 +414723.207}
SPL {X  -162.820, Y  +389.965, Z    +0.000, E1    -3.918, E3 +414722.576}
SPL {X  -162.820, Y  +394.532, Z    +0.000, E1    -7.849, E3 +414724.124}
SPL {X  -162.820, Y  +400.765, Z    +0.000, E1   -14.108, E3 +414721.591}
SPL {X  -162.820, Y  +411.829, Z    +0.000, E1   -24.195, E3 +414723.668}
SPL {X  -162.820, Y  +434.900, Z    +0.000, E1   -34.666, E3 +414751.033}
SPL {X  -162.820, Y  +465.440, Z    +0.000, E1   -41.264, E3 +414792.340}
ENDSPLINE

SPLINE
SPL {X  -162.820, Y  +458.794, Z    +0.000, E1   -36.100, E3 +414805.964}
ENDSPLINE

SPLINE
SPL {X  -162.820, Y  +461.779, Z    +0.000, E1   -35.988, E3 +414815.159}
SPL {X  -162.820, Y  +467.031, Z    +0.000, E1   -36.178, E3 +414829.230}
SPL {X  -162.820, Y  +471.524, Z    +0.000, E1   -36.022, E3 +414842.783}
SPL {X  -162.820, Y  +475.701, Z    +0.000, E1   -36.157, E3 +414853.964}
SPL {X  -162.820, Y  +479.954, Z    +0.000, E1   -36.086, E3 +414866.505}
SPL {X  -162.820, Y  +483.976, Z    +0.000, E1   -36.049, E3 +414878.236}
SPL {X  -162.820, Y  +488.601, Z    +0.000, E1   -36.081, E3 +414891.326}
SPL {X  -162.820, Y  +493.837, Z    +0.000, E1   -36.178, E3 +414905.670}
SPL {X  -162.820, Y  +498.932, Z    +0.000, E1   -36.079, E3 +414920.874}
SPL {X  -162.820, Y  +504.528, Z    +0.000, E1   -36.109, E3 +414936.670}
SPL {X  -162.820, Y  +509.364, Z    +0.000, E1   -36.084, E3 +414950.576}
SPL {X  -162.820, Y  +515.001, Z    +0.000, E1   -36.183, E3 +414966.214}
SPL {X  -162.820, Y  +520.482, Z    +0.000, E1   -36.096, E3 +414982.259}
SPL {X  -162.820, Y  +525.226, Z    +0.000, E1   -36.081, E3 +414995.927}
SPL {X  -162.820, Y  +530.908, Z    +0.000, E1   -36.155, E3 +415011.785}
SPL {X  -162.820, Y  +536.031, Z    +0.000, E1   -36.058, E3 +415026.903}
SPL {X  -162.820, Y  +541.179, Z    +0.000, E1   -36.085, E3 +415041.544}
SPL {X  -162.820, Y  +546.355, Z    +0.000, E1   -36.114, E3 +415056.088}
SPL {X  -162.820, Y  +551.776, Z    +0.000, E1   -36.108, E3 +415071.722}
SPL {X  -162.820, Y  +556.944, Z    +0.000, E1   -36.118, E3 +415086.293}
SPL {X  -162.820, Y  +561.684, Z    +0.000, E1   -36.118, E3 +415099.885}
SPL {X  -162.820, Y  +566.500, Z    +0.000, E1   -36.073, E3 +415113.887}
SPL {X  -162.820, Y  +571.734, Z    +0.000, E1   -36.094, E3 +415128.817}
SPL {X  -162.820, Y  +576.887, Z    +0.000, E1   -36.084, E3 +415143.510}
SPL {X  -162.820, Y  +581.763, Z    +0.000, E1   -36.093, E3 +415157.447}
SPL {X  -162.820, Y  +586.693, Z    +0.000, E1   -36.086, E3 +415171.552}
SPL {X  -162.820, Y  +591.665, Z    +0.000, E1   -36.045, E3 +415186.080}
SPL {X  -162.820, Y  +596.059, Z    +0.000, E1   -36.124, E3 +415198.012}
SPL {X  -162.820, Y  +598.788, Z    +0.000, E1   -36.102, E3 +415205.923}
SPL {X  -162.820, Y  +602.243, Z    +0.000, E1   -36.085, E3 +415215.989}
SPL {X  -162.820, Y  +605.848, Z    +0.000, E1   -36.070, E3 +415226.311}
SPL {X  -162.820, Y  +609.375, Z    +0.000, E1   -36.084, E3 +415236.361}
SPL {X  -162.820, Y  +612.959, Z    +0.000, E1   -36.034, E3 +415246.881}
SPL {X  -162.820, Y  +616.897, Z    +0.000, E1   -36.061, E3 +415258.029}
SPL {X  -162.820, Y  +621.516, Z    +0.000, E1   -36.072, E3 +415271.228}
SPL {X  -162.820, Y  +626.243, Z    +0.000, E1   -36.105, E3 +415284.471}
SPL {X  -162.820, Y  +630.571, Z    +0.000, E1   -36.057, E3 +415297.173}
SPL {X  -162.820, Y  +635.505, Z    +0.000, E1   -36.079, E3 +415311.179}
SPL {X  -162.820, Y  +641.277, Z    +0.000, E1   -36.126, E3 +415327.471}
SPL {X  -162.820, Y  +646.320, Z    +0.000, E1   -36.078, E3 +415342.036}
SPL {X  -162.820, Y  +651.289, Z    +0.000, E1   -36.059, E3 +415356.493}
SPL {X  -162.820, Y  +656.677, Z    +0.000, E1   -36.110, E3 +415371.506}
SPL {X  -162.820, Y  +661.560, Z    +0.000, E1   -36.068, E3 +415385.769}
SPL {X  -162.820, Y  +667.641, Z    +0.000, E1   -36.092, E3 +415403.150}
SPL {X  -162.820, Y  +673.415, Z    +0.000, E1   -36.053, E3 +415419.740}
SPL {X  -162.761, Y  +677.889, Z    +0.000, E1   -36.122, E3 +415432.058}
SPL {X  -162.577, Y  +682.401, Z    +0.000, E1   -36.021, E3 +415445.675}
SPL {X  -162.187, Y  +687.846, Z    +0.000, E1   -36.007, E3 +415461.344}
SPL {X  -161.667, Y  +692.839, Z    +0.000, E1   -35.918, E3 +415476.109}
SPL {X  -161.078, Y  +697.256, Z    +0.000, E1   -35.797, E3 +415489.445}
SPL {X  -160.313, Y  +701.964, Z    +0.000, E1   -35.709, E3 +415503.521}
SPL {X  -159.317, Y  +707.091, Z    +0.000, E1   -35.482, E3 +415519.545}
SPL {X  -158.510, Y  +710.714, Z    +0.000, E1   -35.230, E3 +415531.256}
SPL {X  -155.691, Y  +721.150, Z    +0.000, E1   -39.118, E3 +415536.640}
SPL {X  -154.394, Y  +725.200, Z    +0.000, E1   -39.595, E3 +415543.907}
SPL {X  -152.141, Y  +731.494, Z    +0.000, E1   -35.181, E3 +415599.158}
ENDSPLINE

SPLINE
SPL {X  -160.133, Y  +702.956, Z    +0.000, E1   -19.806, E3 +415642.696}
SPL {X  -161.979, Y  +690.023, Z    +0.000, E1   -12.991, E3 +415645.612}
SPL {X  -162.641, Y  +681.139, Z    +0.000, E1    -7.893, E3 +415647.704}
SPL {X  -162.820, Y  +673.062, Z    +0.000, E1    -2.992, E3 +415646.671}
SPL {X  -162.820, Y  +665.516, Z    +0.000, E1    +2.410, E3 +415648.511}
SPL {X  -162.820, Y  +657.781, Z    +0.000, E1    +9.391, E3 +415646.175}
SPL {X  -162.820, Y  +648.706, Z    +0.000, E1   +17.761, E3 +415647.927}
SPL {X  -162.820, Y  +635.926, Z    +0.000, E1   +28.192, E3 +415652.754}
SPL {X  -162.820, Y  +621.673, Z    +0.000, E1   +34.265, E3 +415669.112}
SPL {X  -162.820, Y  +609.002, Z    +0.000, E1   +38.458, E3 +415682.333}
SPL {X  -162.820, Y  +596.392, Z    +0.000, E1   +37.895, E3 +415715.802}
ENDSPLINE

SPLINE
SPL {X  -162.820, Y  +601.432, Z    +0.000, E1   +34.026, E3 +415725.100}
ENDSPLINE

SPLINE
SPL {X  -162.820, Y  +599.021, Z    +0.000, E1   +33.912, E3 +415733.318}
SPL {X  -162.820, Y  +595.170, Z    +0.000, E1   +33.784, E3 +415746.224}
SPL {X  -162.820, Y  +589.785, Z    +0.000, E1   +33.904, E3 +415762.221}
SPL {X  -162.820, Y  +585.519, Z    +0.000, E1   +33.888, E3 +415775.411}
SPL {X  -162.820, Y  +582.066, Z    +0.000, E1   +33.857, E3 +415786.345}
SPL {X  -162.820, Y  +577.919, Z    +0.000, E1   +33.841, E3 +415799.398}
SPL {X  -162.820, Y  +573.566, Z    +0.000, E1   +33.899, E3 +415812.473}
SPL {X  -162.820, Y  +569.298, Z    +0.000, E1   +33.851, E3 +415826.114}
SPL {X  -162.820, Y  +563.983, Z    +0.000, E1   +33.916, E3 +415842.255}
SPL {X  -162.820, Y  +559.395, Z    +0.000, E1   +33.796, E3 +415857.137}
SPL {X  -162.820, Y  +554.453, Z    +0.000, E1   +33.841, E3 +415872.361}
SPL {X  -162.820, Y  +549.726, Z    +0.000, E1   +33.905, E3 +415886.464}
SPL {X  -162.820, Y  +545.760, Z    +0.000, E1   +33.901, E3 +415898.861}
SPL {X  -162.820, Y  +541.668, Z    +0.000, E1   +33.787, E3 +415912.260}
SPL {X  -162.820, Y  +538.174, Z    +0.000, E1   +33.865, E3 +415922.550}
SPL {X  -162.820, Y  +534.943, Z    +0.000, E1   +33.919, E3 +415932.290}
SPL {X  -162.820, Y  +531.459, Z    +0.000, E1   +33.783, E3 +415943.947}
SPL {X  -162.820, Y  +526.783, Z    +0.000, E1   +33.870, E3 +415958.075}
SPL {X  -162.820, Y  +521.520, Z    +0.000, E1   +33.826, E3 +415974.722}
SPL {X  -162.820, Y  +516.814, Z    +0.000, E1   +33.917, E3 +415988.624}
SPL {X  -162.820, Y  +512.685, Z    +0.000, E1   +33.830, E3 +416002.066}
SPL {X  -162.820, Y  +508.888, Z    +0.000, E1   +33.871, E3 +416013.481}
SPL {X  -162.820, Y  +505.651, Z    +0.000, E1   +33.839, E3 +416023.798}
SPL {X  -162.820, Y  +500.931, Z    +0.000, E1   +34.256, E3 +416035.672}
SPL {X  -162.820, Y  +481.122, Z    +0.000, E1   +41.279, E3 +416045.936}
SPL {X  -162.820, Y  +478.698, Z    +0.000, E1   +40.526, E3 +416056.285}
SPL {X  -162.820, Y  +475.203, Z    +0.000, E1   +39.596, E3 +416070.745}
SPL {X  -162.820, Y  +472.097, Z    +0.000, E1   +38.411, E3 +416085.711}
SPL {X  -162.820, Y  +469.308, Z    +0.000, E1   +37.839, E3 +416096.515}
SPL {X  -162.820, Y  +467.216, Z    +0.000, E1   +37.215, E3 +416106.082}
SPL {X  -162.820, Y  +462.598, Z    +0.000, E1   +37.325, E3 +416118.036}
SPL {X  -162.820, Y  +457.832, Z    +0.000, E1   +37.294, E3 +416131.323}
SPL {X  -162.820, Y  +452.986, Z    +0.000, E1   +37.368, E3 +416144.057}
SPL {X  -162.820, Y  +448.311, Z    +0.000, E1   +37.333, E3 +416157.077}
SPL {X  -162.820, Y  +443.351, Z    +0.000, E1   +37.335, E3 +416170.606}
SPL {X  -162.820, Y  +438.727, Z    +0.000, E1   +37.289, E3 +416183.479}
SPL {X  -162.820, Y  +434.320, Z    +0.000, E1   +37.343, E3 +416195.189}
SPL {X  -162.820, Y  +430.091, Z    +0.000, E1   +37.424, E3 +416206.189}
SPL {X  -162.820, Y  +426.177, Z    +0.000, E1   +37.250, E3 +416218.011}
SPL {X  -162.820, Y  +420.241, Z    +0.000, E1   +37.355, E3 +416233.718}
SPL {X  -162.820, Y  +415.595, Z    +0.000, E1   +37.375, E3 +416246.058}
SPL {X  -162.820, Y  +411.860, Z    +0.000, E1   +37.402, E3 +416256.161}
SPL {X  -162.820, Y  +407.726, Z    +0.000, E1   +37.291, E3 +416268.109}
SPL {X  -162.820, Y  +403.543, Z    +0.000, E1   +37.305, E3 +416279.454}
SPL {X  -162.820, Y  +399.300, Z    +0.000, E1   +37.355, E3 +416290.739}
SPL {X  -162.820, Y  +395.182, Z    +0.000, E1   +37.347, E3 +416302.028}
SPL {X  -162.820, Y  +390.797, Z    +0.000, E1   +37.358, E3 +416313.940}
SPL {X  -162.820, Y  +385.307, Z    +0.000, E1   +37.364, E3 +416329.020}
SPL {X  -162.820, Y  +380.796, Z    +0.000, E1   +37.334, E3 +416341.306}
SPL {X  -162.785, Y  +377.133, Z    +0.000, E1   +37.299, E3 +416351.627}
SPL {X  -162.623, Y  +372.484, Z    +0.000, E1   +37.337, E3 +416364.067}
SPL {X  -162.331, Y  +367.894, Z    +0.000, E1   +37.251, E3 +416377.180}
SPL {X  -161.920, Y  +363.407, Z    +0.000, E1   +37.164, E3 +416389.914}
SPL {X  -161.341, Y  +358.603, Z    +0.000, E1   +37.117, E3 +416403.394}
SPL {X  -160.616, Y  +353.801, Z    +0.000, E1   +36.942, E3 +416417.558}
SPL {X  -159.837, Y  +349.474, Z    +0.000, E1   +36.824, E3 +416430.003}
SPL {X  -159.171, Y  +346.224, Z    +0.000, E1   +36.747, E3 +416439.279}
SPL {X  -158.248, Y  +342.188, Z    +0.000, E1   +36.583, E3 +416451.442}
SPL {X  -153.520, Y  +326.260, Z    +0.000, E1   +41.363, E3 +416464.094}
SPL {X  -150.942, Y  +319.452, Z    +0.000, E1   +36.529, E3 +416520.451}
ENDSPLINE

SPLINE
SPL {X  -159.264, Y  +346.659, Z    +0.000, E1   +22.083, E3 +416561.025}
SPL {X  -161.245, Y  +357.907, Z    +0.000, E1   +16.095, E3 +416574.458}
SPL {X  -162.697, Y  +374.161, Z    +0.000, E1    +7.119, E3 +416572.448}
SPL {X  -162.820, Y  +380.878, Z    +0.000, E1    +2.854, E3 +416575.279}
SPL {X  -162.820, Y  +385.313, Z    +0.000, E1    -0.228, E3 +416575.059}
SPL {X  -162.820, Y  +389.965, Z    +0.000, E1    -3.918, E3 +416574.428}
SPL {X  -162.820, Y  +394.532, Z    +0.000, E1    -7.849, E3 +416575.976}
SPL {X  -162.820, Y  +400.765, Z    +0.000, E1   -14.108, E3 +416573.442}
SPL {X  -162.820, Y  +411.829, Z    +0.000, E1   -24.195, E3 +416575.520}
SPL {X  -162.820, Y  +434.900, Z    +0.000, E1   -34.666, E3 +416602.885}
SPL {X  -162.820, Y  +465.440, Z    +0.000, E1   -41.264, E3 +416644.192}
ENDSPLINE

SPLINE
SPL {X  -162.820, Y  +460.175, Z    +0.000, E1   -36.098, E3 +416661.992}
ENDSPLINE

SPLINE
SPL {X  -162.820, Y  +465.690, Z    +0.000, E1   -36.140, E3 +416677.306}
SPL {X  -162.820, Y  +470.432, Z    +0.000, E1   -36.100, E3 +416691.189}
SPL {X  -162.820, Y  +475.701, Z    +0.000, E1   -36.157, E3 +416705.816}
SPL {X  -162.820, Y  +479.954, Z    +0.000, E1   -36.086, E3 +416718.356}
SPL {X  -162.820, Y  +485.438, Z    +0.000, E1   -36.112, E3 +416734.074}
SPL {X  -162.820, Y  +490.843, Z    +0.000, E1   -36.087, E3 +416749.488}
SPL {X  -162.820, Y  +494.712, Z    +0.000, E1   -36.164, E3 +416760.000}
SPL {X  -162.820, Y  +497.796, Z    +0.000, E1   -36.022, E3 +416769.706}
SPL {X  -162.820, Y  +502.146, Z    +0.000, E1   -36.123, E3 +416781.575}
SPL {X  -162.820, Y  +505.688, Z    +0.000, E1   -36.050, E3 +416792.057}
SPL {X  -162.820, Y  +509.364, Z    +0.000, E1   -36.084, E3 +416802.428}
SPL {X  -162.820, Y  +513.393, Z    +0.000, E1   -36.179, E3 +416813.284}
SPL {X  -162.820, Y  +516.436, Z    +0.000, E1   -36.094, E3 +416822.480}
SPL {X  -162.820, Y  +520.482, Z    +0.000, E1   -36.096, E3 +416834.111}
SPL {X  -162.820, Y  +524.107, Z    +0.000, E1   -36.045, E3 +416844.695}
SPL {X  -162.820, Y  +527.962, Z    +0.000, E1   -36.074, E3 +416855.628}
SPL {X  -162.820, Y  +532.253, Z    +0.000, E1   -36.170, E3 +416867.217}
SPL {X  -162.820, Y  +536.031, Z    +0.000, E1   -36.058, E3 +416878.755}
SPL {X  -162.820, Y  +541.179, Z    +0.000, E1   -36.085, E3 +416893.396}
SPL {X  -162.820, Y  +546.355, Z    +0.000, E1   -36.114, E3 +416907.940}
SPL {X  -162.820, Y  +551.776, Z    +0.000, E1   -36.108, E3 +416923.574}
SPL {X  -162.820, Y  +558.272, Z    +0.000, E1   -36.170, E3 +416941.782}
SPL {X  -162.820, Y  +562.721, Z    +0.000, E1   -36.046, E3 +416955.007}
SPL {X  -162.820, Y  +566.500, Z    +0.000, E1   -36.073, E3 +416965.739}
SPL {X  -162.820, Y  +570.319, Z    +0.000, E1   -36.045, E3 +416976.767}
SPL {X  -162.820, Y  +573.265, Z    +0.000, E1   -36.071, E3 +416985.004}
SPL {X  -162.820, Y  +576.887, Z    +0.000, E1   -36.084, E3 +416995.362}
SPL {X  -162.820, Y  +581.763, Z    +0.000, E1   -36.093, E3 +417009.299}
SPL {X  -162.820, Y  +586.693, Z    +0.000, E1   -36.086, E3 +417023.404}
SPL {X  -162.820, Y  +591.665, Z    +0.000, E1   -36.045, E3 +417037.932}
SPL {X  -162.820, Y  +597.399, Z    +0.000, E1   -36.147, E3 +417053.695}
SPL {X  -162.820, Y  +602.243, Z    +0.000, E1   -36.085, E3 +417067.841}
SPL {X  -162.820, Y  +605.848, Z    +0.000, E1   -36.070, E3 +417078.162}
SPL {X  -162.820, Y  +609.375, Z    +0.000, E1   -36.084, E3 +417088.213}
SPL {X  -162.820, Y  +612.959, Z    +0.000, E1   -36.034, E3 +417098.733}
SPL {X  -162.820, Y  +616.897, Z    +0.000, E1   -36.061, E3 +417109.881}
SPL {X  -162.820, Y  +621.516, Z    +0.000, E1   -36.072, E3 +417123.080}
SPL {X  -162.820, Y  +626.243, Z    +0.000, E1   -36.105, E3 +417136.323}
SPL {X  -162.820, Y  +630.571, Z    +0.000, E1   -36.057, E3 +417149.025}
SPL {X  -162.820, Y  +634.189, Z    +0.000, E1   -36.065, E3 +417159.218}
SPL {X  -162.820, Y  +638.473, Z    +0.000, E1   -36.098, E3 +417171.455}
SPL {X  -162.820, Y  +642.832, Z    +0.000, E1   -36.091, E3 +417183.781}
SPL {X  -162.820, Y  +646.320, Z    +0.000, E1   -36.078, E3 +417193.888}
SPL {X  -162.820, Y  +649.997, Z    +0.000, E1   -36.000, E3 +417204.859}
SPL {X  -162.820, Y  +655.571, Z    +0.000, E1   -36.141, E3 +417220.193}
SPL {X  -162.820, Y  +661.560, Z    +0.000, E1   -36.068, E3 +417237.621}
SPL {X  -162.820, Y  +667.641, Z    +0.000, E1   -36.092, E3 +417255.002}
SPL {X  -162.820, Y  +673.415, Z    +0.000, E1   -36.053, E3 +417271.592}
SPL {X  -162.761, Y  +677.889, Z    +0.000, E1   -36.122, E3 +417283.910}
SPL {X  -162.577, Y  +682.401, Z    +0.000, E1   -36.021, E3 +417297.527}
SPL {X  -162.187, Y  +687.846, Z    +0.000, E1   -36.007, E3 +417313.196}
SPL {X  -161.667, Y  +692.839, Z    +0.000, E1   -35.918, E3 +417327.961}
SPL {X  -161.078, Y  +697.256, Z    +0.000, E1   -35.797, E3 +417341.297}
SPL {X  -160.313, Y  +701.964, Z    +0.000, E1   -35.709, E3 +417355.372}
SPL {X  -159.317, Y  +707.091, Z    +0.000, E1   -35.482, E3 +417371.396}
SPL {X  -158.510, Y  +710.714, Z    +0.000, E1   -35.230, E3 +417383.107}
SPL {X  -155.037, Y  +723.239, Z    +0.000, E1   -39.382, E3 +417392.204}
SPL {X  -152.141, Y  +731.494, Z    +0.000, E1   -35.181, E3 +417451.010}
ENDSPLINE

